// TwinCAT 3 PLC project CFFwelding
// ProgramVersion: 3.1.4024.0
// libraries:
//   Tc2_Standard, * (Beckhoff Automation GmbH)
//   Tc2_System, * (Beckhoff Automation GmbH)
//   Tc3_Module, * (Beckhoff Automation GmbH)
//   Tc2_MC2,3.3.65.0,Beckhoff Automation GmbH
// project tree:
//   Tasks/ Task_CffFast.TcTTO, Task_CffMain.TcTTO, Task_CffSlow.TcTTO
//   DUTs/Enums/ E_OperationMode.TcDUT, E_ControlSource.TcDUT, E_MachineState.TcDUT (not stored), E_InitializeState.TcDUT, E_MaintenanceFunction.TcDUT (not stored), E_MaintenanceState.TcDUT, E_CffState.TcDUT (not stored), E_CffExitIntent.TcDUT, E_CffStep.TcDUT, E_StepSubPhase.TcDUT, E_StepPrimaryCriterion.TcDUT, E_SecondaryCriterionAction.TcDUT, E_StepEndCause.TcDUT, E_ZCommandOwner.TcDUT, E_ZExtSetpointState.TcDUT (not stored), E_ZExternalTrajectoryState.TcDUT (not stored), E_AlarmLevel.TcDUT, E_AlarmCode.TcDUT (not stored), E_FastenerStatus.TcDUT, E_FeederState.TcDUT, E_ReturnMode.TcDUT, E_CalibrationState.TcDUT, E_CommandExecutionState.TcDUT, E_CommandRejectReason.TcDUT (not stored), E_HmiCommandCode.TcDUT, E_RobotCommandCode.TcDUT, E_ProgramState.TcDUT, E_InterfaceEventState.TcDUT
//   DUTs/Structures/ ST_MachineConfig.TcDUT (not stored), ST_MachineLimits.TcDUT (not stored), ST_ForceCalibration.TcDUT (not stored), ST_DisplacementCalibration.TcDUT, ST_CollisionCalibration.TcDUT (not stored), ST_ZForceControlProfile.TcDUT, ST_RAxisProfile.TcDUT (not stored), ST_StepProceedingConfig.TcDUT, ST_CffStepProgram.TcDUT (not stored), ST_JoinProgramHeader.TcDUT (not stored), ST_ProcessMonitorProfile.TcDUT, ST_CffJoinProgram.TcDUT (not stored), ST_JoiningPointAssignment.TcDUT, ST_CycleSnapshot.TcDUT, ST_ProcessActual.TcDUT (not stored), ST_ProcessFeatures.TcDUT, ST_StepCriterionResult.TcDUT, ST_CycleResult.TcDUT, ST_AlarmRequest.TcDUT (not stored), ST_AlarmStatus.TcDUT, ST_CommandMailbox.TcDUT, ST_CommandPermission.TcDUT, ST_MaintenanceHoldRequest.TcDUT, ST_RobotCommand.TcDUT (not stored), ST_RobotStatus.TcDUT, ST_FeederInput.TcDUT (not stored), ST_FeederOutput.TcDUT, ST_CalibrationCommand.TcDUT (not stored), ST_CalibrationStatus.TcDUT, ST_FastCommand.TcDUT (not stored), ST_FastStatus.TcDUT, ST_CurveSample.TcDUT, ST_HardwareBindingStatus.TcDUT (not stored), ST_SensorProcessingConfig.TcDUT (not stored), ST_ZExtSetpointConfig.TcDUT, ST_CffSequenceConfig.TcDUT, ST_CffFastConfigSnapshot.TcDUT (not stored)
//   GVLs/ GVL_Const.TcGVL (not stored), GVL_IO.TcGVL, GVL_Config.TcGVL, GVL_Calibration.TcGVL, GVL_Program.TcGVL, GVL_Command.TcGVL, GVL_Status.TcGVL, GVL_Process.TcGVL, GVL_Alarm.TcGVL, GVL_HMI.TcGVL (not stored), GVL_Trace.TcGVL, GVL_Persistent.TcGVL, GVL_ProjectInfo.TcGVL (not stored), GVL_FastInternal.TcGVL
//   DUTs/Interfaces/ ST_ZForceControlInput.TcDUT (not stored), ST_ZForceControlOutput.TcDUT, ST_ZExtSetpointCommand.TcDUT (not stored), ST_ZExtSetpointStatus.TcDUT, ST_ZAxisCommand.TcDUT, ST_ZAxisStatus.TcDUT, ST_RAxisCommand.TcDUT, ST_RAxisStatus.TcDUT (not stored), ST_CffMotionIntent.TcDUT (not stored), ST_ZExternalTrajectoryInput.TcDUT (not stored), ST_ZExternalTrajectoryOutput.TcDUT, ST_ContactDetectInput.TcDUT, ST_ContactDetectOutput.TcDUT, ST_ForceDeclineInput.TcDUT, ST_ForceDeclineOutput.TcDUT, ST_StepCriterionInput.TcDUT (not stored), ST_StepCriterionOutput.TcDUT, ST_CffSequenceCommand.TcDUT, ST_CffSequenceStatus.TcDUT (not stored), ST_ProcessReferenceCommand.TcDUT (not stored)
//   POUs/Functions/ FC_ClampLReal.TcPOU, FC_ScaleLinear.TcPOU (not stored), FC_LimitRate.TcPOU, FC_TrapezoidIntegrate.TcPOU (not stored), FC_RpmToRadPerSec.TcPOU (not stored), FC_CalcEnergyIncrement.TcPOU, FC_ConvertDirection.TcPOU, FC_IsFiniteLReal.TcPOU, FC_IsNewerRequestId.TcPOU (not stored), FC_ValidateCffSequenceConfig.TcPOU (not stored), FC_Interpolate1D.TcPOU, FC_ValidateCalibration.TcPOU, FC_ValidateJoinProgram.TcPOU, FC_GetPrimaryEndCause.TcPOU (not stored), FC_CalcStrokeVelocityLimit.TcPOU, FC_CheckModeSourceMatrix.TcPOU
//   POUs/FunctionBlocks/Utility/ FB_LowPassFilter.TcPOU, FB_Debounce.TcPOU (not stored), FB_SignalValidity.TcPOU (not stored), FB_SetpointRamp.TcPOU, FB_CommandHandshake.TcPOU, FB_AlarmLatch.TcPOU
//   POUs/FunctionBlocks/Axis/ FB_AxisCommandArbiter.TcPOU, FB_ZAxisNcAdapter.TcPOU, FB_RAxisNcAdapter.TcPOU, FB_ZAxisExtSetpointAdapter.TcPOU
//   POUs/FunctionBlocks/Control/ FB_BumplessProfileSwitch.TcPOU, FB_ZForceAdmittance.TcPOU, FB_ZExternalTrajectory.TcPOU, FB_ContactDetect.TcPOU (not stored), FB_ForceDeclineObserver.TcPOU, FB_StepProceedingCriterion.TcPOU
//   POUs/Fast/ PRG_FastInputs.TcPOU, PRG_CffSequence.TcPOU, PRG_FastAxisControl.TcPOU, PRG_FastMonitoring.TcPOU
//   POUs/Main/ PRG_ModeControl.TcPOU, PRG_RobotInterface.TcPOU (not stored), PRG_CommandDispatcher.TcPOU, PRG_ProgramManager.TcPOU, PRG_InitializeControl.TcPOU, PRG_ServiceCalibration.TcPOU (not stored), PRG_MaintenanceControl.TcPOU, PRG_ManualControl.TcPOU (not stored), PRG_AutoControl.TcPOU, PRG_FastenerControl.TcPOU, PRG_FeederControl.TcPOU, PRG_ClampControl.TcPOU (not stored), PRG_MachineMain.TcPOU (not stored), PRG_AlarmControl.TcPOU, PRG_TowerLightControl.TcPOU (not stored)
//   POUs/Slow/ PRG_HmiAdsInterface.TcPOU (not stored), PRG_ResultTraceability.TcPOU (not stored), PRG_Statistics.TcPOU, PRG_Persistence.TcPOU (not stored)
// real-time tasks:
//   TASK Task_CffMain: cycle T#10ms, priority 20, ADS port 350
//   TASK Task_CffFast: cycle T#2ms, priority 10, ADS port 351
//   TASK Task_CffSlow: cycle T#50000us, priority 30, ADS port 352
// motion (NC):
//   TASK NC_Cff SAF: cycle T#2ms, priority 4, ADS port 501
//   TASK NC_Cff SVB: cycle T#10ms, priority 8, ADS port 511
//   AXIS Z_Axis_NC (id 1)
//     OtherSettings: AllowMotionCmdToSlave=true
//     encoder EncType=1
//     drive DrvType=5
//       Analog: TorqueSetpointScale=10, ScaleFactorActTorque=0.1
//       TimeComp: TaskDelayCycles=1
//     controller CtrType=1
//       CtrPara: PriorControlFactor=1
//         Observer: BandWidth=20
//   AXIS R_Axis_NC (id 2)
//     OtherSettings: AllowMotionCmdToSlave=true
//     encoder EncType=1
//     drive DrvType=5
//       Analog: TorqueSetpointScale=10, ScaleFactorActTorque=0.1
//       TimeComp: TaskDelayCycles=1
//     controller CtrType=1
//       CtrPara: PriorControlFactor=1
//         Observer: BandWidth=20
// variable links:
//   CFFwelding/CFFwelding Instance <-> NC_Cff SAF/Axes/R_Axis_NC
//     Task_CffFast Inputs/GVL_IO.R_axis.NcToPlc <-> Outputs/ToPlc
//     Task_CffFast Outputs/GVL_IO.R_axis.PlcToNc <-> Inputs/FromPlc
//   CFFwelding/CFFwelding Instance <-> NC_Cff SAF/Axes/Z_Axis_NC
//     Task_CffFast Inputs/GVL_IO.Z_axis.NcToPlc <-> Outputs/ToPlc
//     Task_CffFast Outputs/GVL_IO.Z_axis.PlcToNc <-> Inputs/FromPlc

CONFIGURATION CFFwelding
    RESOURCE PLC ON TwinCAT3
        TASK Task_CffFast(INTERVAL := T#2ms, PRIORITY := 10);
        TASK Task_CffMain(INTERVAL := T#10ms, PRIORITY := 20);
        TASK Task_CffSlow(INTERVAL := T#50000us, PRIORITY := 30);
        PROGRAM PRG_FastInputs WITH Task_CffFast : PRG_FastInputs;
        PROGRAM PRG_CffSequence WITH Task_CffFast : PRG_CffSequence;
        PROGRAM PRG_FastAxisControl WITH Task_CffFast : PRG_FastAxisControl;
        PROGRAM PRG_FastMonitoring WITH Task_CffFast : PRG_FastMonitoring;
        PROGRAM PRG_ModeControl WITH Task_CffMain : PRG_ModeControl;
        PROGRAM PRG_RobotInterface WITH Task_CffMain : PRG_RobotInterface;
        PROGRAM PRG_CommandDispatcher WITH Task_CffMain : PRG_CommandDispatcher;
        PROGRAM PRG_ProgramManager WITH Task_CffMain : PRG_ProgramManager;
        PROGRAM PRG_InitializeControl WITH Task_CffMain : PRG_InitializeControl;
        PROGRAM PRG_ServiceCalibration WITH Task_CffMain : PRG_ServiceCalibration;
        PROGRAM PRG_MaintenanceControl WITH Task_CffMain : PRG_MaintenanceControl;
        PROGRAM PRG_ManualControl WITH Task_CffMain : PRG_ManualControl;
        PROGRAM PRG_AutoControl WITH Task_CffMain : PRG_AutoControl;
        PROGRAM PRG_FastenerControl WITH Task_CffMain : PRG_FastenerControl;
        PROGRAM PRG_FeederControl WITH Task_CffMain : PRG_FeederControl;
        PROGRAM PRG_ClampControl WITH Task_CffMain : PRG_ClampControl;
        PROGRAM PRG_MachineMain WITH Task_CffMain : PRG_MachineMain;
        PROGRAM PRG_AlarmControl WITH Task_CffMain : PRG_AlarmControl;
        PROGRAM PRG_TowerLightControl WITH Task_CffMain : PRG_TowerLightControl;
        PROGRAM PRG_HmiAdsInterface WITH Task_CffSlow : PRG_HmiAdsInterface;
        PROGRAM PRG_ResultTraceability WITH Task_CffSlow : PRG_ResultTraceability;
        PROGRAM PRG_Statistics WITH Task_CffSlow : PRG_Statistics;
        PROGRAM PRG_Persistence WITH Task_CffSlow : PRG_Persistence;
    END_RESOURCE
END_CONFIGURATION

// ---- DUTs/Enums/E_OperationMode.TcDUT
TYPE E_OperationMode : (
    OP_MODE_INVALID := 0,
    OP_MODE_MAINTENANCE := 10,
    OP_MODE_MANUAL := 20,
    OP_MODE_AUTOMATIC := 30
); END_TYPE

// ---- DUTs/Enums/E_ControlSource.TcDUT
TYPE E_ControlSource : (
    CONTROL_SOURCE_INVALID := 0,
    CONTROL_SOURCE_LOCAL := 10,
    CONTROL_SOURCE_ROBOT := 20
); END_TYPE

// ---- DUTs/Enums/E_InitializeState.TcDUT
TYPE E_InitializeState : (
    INIT_IDLE := 0,
    INIT_CLEAR_TRANSIENTS := 10,
    INIT_VALIDATE_MODE_SOURCE := 20,
    INIT_VALIDATE_COMMUNICATION := 30,
    INIT_VALIDATE_SENSORS := 40,
    INIT_RESET_AXIS_ERRORS := 50,
    INIT_HOME_Z_IF_REQUIRED := 60,
    INIT_HOME_R_IF_REQUIRED := 70,
    INIT_STOP_R := 80,
    INIT_RETURN_Z_REFERENCE := 90,
    INIT_RETURN_CYLINDERS := 100,
    INIT_RESET_FEEDER := 110,
    INIT_VALIDATE_CALIBRATIONS := 120,
    INIT_VALIDATE_ACTIVE_PROGRAM := 130,
    INIT_FINAL_READY_CHECK := 140,
    INIT_COMPLETE := 150,
    INIT_FAILED := 200
); END_TYPE

// ---- DUTs/Enums/E_MaintenanceState.TcDUT
TYPE E_MaintenanceState : (
    MAINT_STATE_IDLE := 0,
    MAINT_STATE_SELECTED := 10,
    MAINT_STATE_PRECHECK := 20,
    MAINT_STATE_ACTIVE := 30,
    MAINT_STATE_STOPPING := 40,
    MAINT_STATE_COMPLETE := 50,
    MAINT_STATE_CANCELLED := 60,
    MAINT_STATE_FAULT := 100
); END_TYPE

// ---- DUTs/Enums/E_CffExitIntent.TcDUT
TYPE E_CffExitIntent : (
    CFF_EXIT_NONE := 0,
    CFF_EXIT_NORMAL_RETURN := 10,
    CFF_EXIT_NOK_RETURN := 20,
    CFF_EXIT_ABORT_NO_RETURN := 30,
    CFF_EXIT_FAULT_NO_RETURN := 40
); END_TYPE

// ---- DUTs/Enums/E_CffStep.TcDUT
TYPE E_CffStep : (
    CFF_STEP_NONE := 0,
    CFF_STEP1_PENETRATION := 10,
    CFF_STEP2_CLEAN_ACTIVATE := 20,
    CFF_STEP3_WELDING := 30,
    CFF_STEP4_COMPRESSION := 40
); END_TYPE

// ---- DUTs/Enums/E_StepSubPhase.TcDUT
TYPE E_StepSubPhase : (
    STEP_SUBPHASE_NONE := 0,
    STEP_SUBPHASE_ENTRY := 10,
    STEP_SUBPHASE_RAMP_PROCESS := 20,
    STEP_SUBPHASE_END_CHECK := 30,
    STEP_SUBPHASE_BRAKE_COMPRESSION := 40,
    STEP_SUBPHASE_VALID_FORCE_HOLD := 50
); END_TYPE

// ---- DUTs/Enums/E_StepPrimaryCriterion.TcDUT
TYPE E_StepPrimaryCriterion : (
    STEP_CRIT_RELATIVE_DISTANCE := 0,
    STEP_CRIT_STEP_TIME := 10,
    STEP_CRIT_FORCE_DECLINE_TO := 20
); END_TYPE

// ---- DUTs/Enums/E_SecondaryCriterionAction.TcDUT
TYPE E_SecondaryCriterionAction : (
    SECONDARY_ADVANCE_AND_NOK := 0,
    SECONDARY_CONTROLLED_EXIT_NOK := 10
); END_TYPE

// ---- DUTs/Enums/E_StepEndCause.TcDUT
TYPE E_StepEndCause : (
    STEP_END_NONE := 0,
    STEP_END_PRIMARY_RELATIVE_DISTANCE := 10,
    STEP_END_PRIMARY_STEP_TIME := 20,
    STEP_END_PRIMARY_FORCE_DECLINE := 30,
    STEP_END_SECONDARY_RELATIVE_DISTANCE := 40,
    STEP_END_MAX_TIME := 50,
    STEP_END_HARD_FORCE := 60,
    STEP_END_HARD_STROKE := 70,
    STEP_END_COLLISION := 110,
    STEP_END_SENSOR_INVALID := 80,
    STEP_END_AXIS_FAULT := 90,
    STEP_END_STOP_REQUEST := 100
); END_TYPE

// ---- DUTs/Enums/E_ZCommandOwner.TcDUT
TYPE E_ZCommandOwner : (
    Z_OWNER_NONE := 0,
    Z_OWNER_HOME := 10,
    Z_OWNER_MANUAL := 20,
    Z_OWNER_APPROACH := 30,
    Z_OWNER_FORCE_PROCESS := 40,
    Z_OWNER_RETRACT := 50,
    Z_OWNER_FAULT_STOP := 100
); END_TYPE

// ---- DUTs/Enums/E_AlarmLevel.TcDUT
TYPE E_AlarmLevel : (
    ALARM_LEVEL_NONE := 0,
    ALARM_LEVEL_WARNING := 10,
    ALARM_LEVEL_NOK := 20,
    ALARM_LEVEL_FAULT := 30
); END_TYPE

// ---- DUTs/Enums/E_FastenerStatus.TcDUT
TYPE E_FastenerStatus : (
    FASTENER_UNKNOWN := 0,
    FASTENER_EMPTY := 10,
    FASTENER_SINGLE_OK := 20,
    FASTENER_WRONG_TYPE := 30,
    FASTENER_MULTIPLE := 40,
    FASTENER_JAMMED := 50,
    FASTENER_FAULT := 100
); END_TYPE

// ---- DUTs/Enums/E_FeederState.TcDUT
TYPE E_FeederState : (
    FEEDER_IDLE := 0,
    FEEDER_REQUEST := 10,
    FEEDER_FEEDING := 20,
    FEEDER_VERIFY := 30,
    FEEDER_COMPLETE := 40,
    FEEDER_FAULT := 100
); END_TYPE

// ---- DUTs/Enums/E_ReturnMode.TcDUT
TYPE E_ReturnMode : (
    RETURN_MODE_LOCAL := 0,
    RETURN_MODE_REFERENCE := 10
); END_TYPE

// ---- DUTs/Enums/E_CalibrationState.TcDUT
TYPE E_CalibrationState : (
    CAL_STATE_IDLE := 0,
    CAL_STATE_PRECHECK := 10,
    CAL_STATE_ACTIVE := 20,
    CAL_STATE_VALIDATE := 30,
    CAL_STATE_COMPLETE := 40,
    CAL_STATE_FAILED := 100
); END_TYPE

// ---- DUTs/Enums/E_CommandExecutionState.TcDUT
TYPE E_CommandExecutionState : (
    COMMAND_IDLE := 0,
    COMMAND_ACCEPTED := 10,
    COMMAND_EXECUTING := 20,
    COMMAND_COMPLETED := 30,
    COMMAND_REJECTED := 40,
    COMMAND_FAILED := 50,
    COMMAND_CANCELLED := 60
); END_TYPE

// ---- DUTs/Enums/E_HmiCommandCode.TcDUT
TYPE E_HmiCommandCode : (
    HMI_CMD_NONE := 0,
    HMI_CMD_START := 10,
    HMI_CMD_STOP := 20,
    HMI_CMD_INITIALIZE := 30,
    HMI_CMD_RESET := 40,
    HMI_CMD_ACK_RESULT := 50,
    HMI_CMD_SELECT_MAINTENANCE := 60,
    HMI_CMD_EXECUTE_MAINTENANCE := 70,
    HMI_CMD_CANCEL_MAINTENANCE := 80,
    HMI_CMD_VALIDATE_STEP := 90,
    HMI_CMD_SAVE_STEP := 100,
    HMI_CMD_VALIDATE_PROGRAM := 110,
    HMI_CMD_SAVE_PROGRAM := 120,
    HMI_CMD_ACTIVATE_PROGRAM := 130,
    HMI_CMD_SAVE_JOINING_POINT := 140,
    HMI_CMD_REQUEST_ALARM_PAGE := 150,
    HMI_CMD_REQUEST_CURVE_PAGE := 160
); END_TYPE

// ---- DUTs/Enums/E_RobotCommandCode.TcDUT
TYPE E_RobotCommandCode : (
    ROBOT_CMD_NONE := 0,
    ROBOT_CMD_START := 10,
    ROBOT_CMD_STOP := 20,
    ROBOT_CMD_INITIALIZE := 30,
    ROBOT_CMD_RESET := 40,
    ROBOT_CMD_ABORT := 50
); END_TYPE

// ---- DUTs/Enums/E_ProgramState.TcDUT
TYPE E_ProgramState : (
    PROGRAM_EMPTY := 0,
    PROGRAM_DRAFT := 10,
    PROGRAM_VALID := 20,
    PROGRAM_ACTIVE := 30,
    PROGRAM_INVALID := 40
); END_TYPE

// ---- DUTs/Enums/E_InterfaceEventState.TcDUT
TYPE E_InterfaceEventState : (
    INTERFACE_EVENT_IDLE := 0,
    INTERFACE_EVENT_CANDIDATE := 10,
    INTERFACE_EVENT_CONFIRMED := 20,
    INTERFACE_EVENT_REJECTED := 30,
    INTERFACE_EVENT_EXPIRED := 40
); END_TYPE

// ---- DUTs/Structures/ST_DisplacementCalibration.TcDUT
TYPE ST_DisplacementCalibration : STRUCT
    (* 位移传感器零点原始值。 *)
    fRawZero : LREAL;
    (* 原始值至毫米的增益。 *)
    fGainMmPerCount : LREAL;
    (* 位移零点偏置，单位毫米。 *)
    fOffsetMm : LREAL;
    (* 位移方向系数，仅允许正一或负一。 *)
    nDirection : DINT;
    (* 标定最大残差，单位毫米。 *)
    fMaxResidualMm : LREAL;
    (* 标定修订号。 *)
    nRevision : UDINT;
    (* 标定数据是否有效。 *)
    bValid : BOOL;
END_STRUCT
END_TYPE

// ---- DUTs/Structures/ST_ZForceControlProfile.TcDUT
TYPE ST_ZForceControlProfile : STRUCT
    (* Profile编号。 *)
    nProfileId : UDINT;
    (* Profile修订号；变化时必须执行积分无扰预置。 *)
    nRevision : UDINT;
    (* 速度前馈，向下为正，单位毫米每秒。 *)
    fVelocityFeedForwardMmS : LREAL;
    (* 比例增益，单位毫米每秒每千牛。 *)
    fKp : LREAL;
    (* 积分增益，单位毫米每二次方秒每千牛。 *)
    fKi : LREAL;
    (* 抗积分饱和回算增益，单位每秒。 *)
    fKaw : LREAL;
    (* 积分项绝对限幅，单位毫米每秒。 *)
    fIntegralLimit : LREAL;
    (* 向上最大速度，单位毫米每秒。 *)
    fMaxUpVelocityMmS : LREAL;
    (* 向下最大速度，单位毫米每秒。 *)
    fMaxDownVelocityMmS : LREAL;
    (* 最大加速度，单位毫米每二次方秒。 *)
    fMaxAccelerationMmS2 : LREAL;
    (* 制动距离裕量，单位毫米。 *)
    fBrakeMarginMm : LREAL;
    (* 设定力斜坡，单位牛顿每秒。 *)
    fForceRampNS : LREAL;
    (* 参数是否有效。 *)
    bValid : BOOL;
END_STRUCT
END_TYPE

// ---- DUTs/Structures/ST_StepProceedingConfig.TcDUT
TYPE ST_StepProceedingConfig : STRUCT
    (* 本步骤唯一主结束判据。 *)
    ePrimaryCriterion : E_StepPrimaryCriterion;
    (* 次级判据触发后的动作。 *)
    eSecondaryAction : E_SecondaryCriterionAction;
    (* 相对位移阈值，单位毫米。 *)
    fRelativeDistanceMm : LREAL;
    (* Step Time主判据目标，单位毫秒。 *)
    nPrimaryStepTimeMs : UDINT;
    (* 步骤质量最短时间，单位毫秒。 *)
    nStepMinMs : UDINT;
    (* Primary等待看门狗时间，单位毫秒。 *)
    nStepMaxMs : UDINT;
    (* Time或Decline主判据使用的累计S_rel次级边界，单位毫米。 *)
    fSecondarySRelMm : LREAL;
    (* 力下降确认阈值，单位牛顿。 *)
    fDeclineToN : LREAL;
    (* 力下降观察武装阈值，单位牛顿。 *)
    fArmForceN : LREAL;
    (* 力下降确认回差，单位牛顿。 *)
    fDeclineHysteresisN : LREAL;
    (* 力下降最小变化率绝对值，单位牛顿每秒。 *)
    fMinimumDeclineRateNS : LREAL;
    (* 力下降连续确认时间，单位毫秒。 *)
    nDeclineDebounceMs : UDINT;
    (* 力下降判据有效S_rel窗口下限，单位毫米。 *)
    fCriterionSRelMinMm : LREAL;
    (* 力下降判据有效S_rel窗口上限，单位毫米。 *)
    fCriterionSRelMaxMm : LREAL;
    (* 力下降判据最小主轴转速绝对值，单位转每分钟。 *)
    fCriterionRpmMin : LREAL;
    (* 判据允许的最大Z轴捕获速度绝对值，单位毫米每秒。 *)
    fCaptureMaxVelocityMmS : LREAL;
    (* 合格力带连续保持时间，单位毫秒。 *)
    nQualifiedForceHoldMs : UDINT;
    (* 合格力带容差，单位牛顿。 *)
    fForceBandToleranceN : LREAL;
    (* R轴停止阈值，单位转每分钟。 *)
    fRpmStoppedThresholdRpm : LREAL;
    (* 判据配置是否有效。 *)
    bValid : BOOL;
END_STRUCT
END_TYPE

// ---- DUTs/Structures/ST_ProcessMonitorProfile.TcDUT
TYPE ST_ProcessMonitorProfile : STRUCT
    (* 最小允许过程力，单位牛顿。 *)
    fMinForceN : LREAL;
    (* 最大允许过程力，单位牛顿。 *)
    fMaxForceN : LREAL;
    (* 最小允许相对位移，单位毫米。 *)
    fMinRelativeDistanceMm : LREAL;
    (* 最大允许相对位移，单位毫米。 *)
    fMaxRelativeDistanceMm : LREAL;
    (* 最小允许扭矩，单位牛米。 *)
    fMinTorqueNm : LREAL;
    (* 最大允许扭矩，单位牛米。 *)
    fMaxTorqueNm : LREAL;
    (* 最小允许能量，单位焦耳。 *)
    fMinEnergyJ : LREAL;
    (* 最大允许能量，单位焦耳。 *)
    fMaxEnergyJ : LREAL;
    (* 监控参数是否有效。 *)
    bValid : BOOL;
END_STRUCT
END_TYPE

// ---- DUTs/Structures/ST_JoiningPointAssignment.TcDUT
TYPE ST_JoiningPointAssignment : STRUCT
    (* 机器人加工点编号。 *)
    nJoiningPointId : UDINT;
    (* 该点关联的加工程序编号。 *)
    nProgramId : UDINT;
    (* 关联关系修订号。 *)
    nRevision : UDINT;
    (* 关联关系是否有效。 *)
    bValid : BOOL;
END_STRUCT
END_TYPE

// ---- DUTs/Structures/ST_CycleSnapshot.TcDUT
TYPE ST_CycleSnapshot : STRUCT
    (* 周期请求编号。 *)
    nRequestId : UDINT;
    (* 已接受的加工点编号。 *)
    nJoiningPointId : UDINT;
    (* 已冻结的加工程序。 *)
    stProgram : ST_CffJoinProgram;
    (* 机器配置修订号。 *)
    nMachineConfigRevision : UDINT;
    (* 标定修订号。 *)
    nCalibrationRevision : UDINT;
    (* 快照修订号。 *)
    nSnapshotRevision : UDINT;
    (* 快照完整性校验值。 *)
    nCrc32 : UDINT;
    (* 周期快照是否可执行。 *)
    bValid : BOOL;
END_STRUCT
END_TYPE

// ---- DUTs/Structures/ST_ProcessFeatures.TcDUT
TYPE ST_ProcessFeatures : STRUCT
    (* 周期最大力，单位牛顿。 *)
    fMaxForceN : LREAL;
    (* 周期平均力，单位牛顿。 *)
    fMeanForceN : LREAL;
    (* 周期最大扭矩，单位牛米。 *)
    fMaxTorqueNm : LREAL;
    (* 周期平均扭矩，单位牛米。 *)
    fMeanTorqueNm : LREAL;
    (* 周期最终相对位移，单位毫米。 *)
    fFinalRelativeDistanceMm : LREAL;
    (* 周期累计能量，单位焦耳。 *)
    fEnergyJ : LREAL;
    (* 有效采样数量。 *)
    nSampleCount : UDINT;
    (* 特征提取结果是否有效。 *)
    bValid : BOOL;
END_STRUCT
END_TYPE

// ---- DUTs/Structures/ST_StepCriterionResult.TcDUT
TYPE ST_StepCriterionResult : STRUCT
    (* 被评估的 CFF 步骤。 *)
    eStep : E_CffStep;
    (* 实际步骤结束原因。 *)
    eEndCause : E_StepEndCause;
    (* 主判据是否已经锁存。 *)
    bPrimaryLatched : BOOL;
    (* 次级判据是否已经锁存。 *)
    bSecondaryLatched : BOOL;
    (* 步骤是否判为不合格。 *)
    bNok : BOOL;
    (* 判据触发时的周期计数。 *)
    nTriggerCycle : UDINT;
    (* 步骤是否过短。 *)
    bTooShort : BOOL;
    (* 合格力带保持时间是否满足。 *)
    bQualifiedForceHoldMet : BOOL;
    (* 合格力带实际保持时间，单位秒。 *)
    rQualifiedForceHoldTime_s : LREAL;
    (* 锁存的轴向力，单位千牛。 *)
    rLatchedForce_kN : LREAL;
    (* 锁存的相对位置，单位毫米。 *)
    rLatchedRelativePosition_mm : LREAL;
    (* 锁存的步骤时间，单位秒。 *)
    rLatchedStepTime_s : LREAL;
END_STRUCT
END_TYPE

// ---- DUTs/Structures/ST_CycleResult.TcDUT
TYPE ST_CycleResult : STRUCT
    (* 全局焊接结果编号。 *)
    nWeldId : ULINT;
    (* 加工点编号。 *)
    nJoiningPointId : UDINT;
    (* 加工程序编号。 *)
    nProgramId : UDINT;
    (* 周期是否合格。 *)
    bOk : BOOL;
    (* 周期是否不合格。 *)
    bNok : BOOL;
    (* 周期是否中止。 *)
    bAborted : BOOL;
    (* 四个步骤的实际结束原因。 *)
    aeStepEndCause : ARRAY[1..4] OF E_StepEndCause;
    (* 周期特征值。 *)
    stFeatures : ST_ProcessFeatures;
    (* 周期持续时间，单位毫秒。 *)
    nCycleTimeMs : UDINT;
    (* 曲线缓冲区是否完整。 *)
    bCurveBufferComplete : BOOL;
    (* 已记录的曲线样本数量。 *)
    nCurveSampleCount : UDINT;
END_STRUCT
END_TYPE

// ---- DUTs/Structures/ST_AlarmStatus.TcDUT
TYPE ST_AlarmStatus : STRUCT
    (* 当前最高优先级报警代码。 *)
    eCurrentCode : E_AlarmCode;
    (* 当前最高报警等级。 *)
    eCurrentLevel : E_AlarmLevel;
    (* 是否存在活动报警。 *)
    bActive : BOOL;
    (* 当前报警是否已确认。 *)
    bAcknowledged : BOOL;
    (* 活动报警数量。 *)
    nActiveCount : UINT;
    (* 报警集合修订号。 *)
    nRevision : UDINT;
END_STRUCT
END_TYPE

// ---- DUTs/Structures/ST_CommandMailbox.TcDUT
TYPE ST_CommandMailbox : STRUCT
    (* 单调递增的命令请求编号。 *)
    nRequestId : UDINT;
    (* 控制源类型。 *)
    eSource : E_ControlSource;
    (* HMI 命令代码。 *)
    eHmiCommand : E_HmiCommandCode;
    (* 机器人命令代码。 *)
    eRobotCommand : E_RobotCommandCode;
    (* 命令目标对象编号。 *)
    nObjectId : UDINT;
    (* 通用整数载荷。 *)
    nPayloadDint : DINT;
    (* 通用浮点载荷。 *)
    fPayloadLreal : LREAL;
    (* 命令执行状态。 *)
    eState : E_CommandExecutionState;
    (* 命令拒绝原因。 *)
    eRejectReason : E_CommandRejectReason;
END_STRUCT
END_TYPE

// ---- DUTs/Structures/ST_CommandPermission.TcDUT
TYPE ST_CommandPermission : STRUCT
    (* 是否允许启动自动周期。 *)
    bAllowCycleStart : BOOL;
    (* 是否允许复位故障。 *)
    bAllowReset : BOOL;
    (* 是否允许手动 Z 轴动作。 *)
    bAllowManualZ : BOOL;
    (* 是否允许手动 R 轴动作。 *)
    bAllowManualR : BOOL;
    (* 是否允许执行维护功能。 *)
    bAllowMaintenance : BOOL;
    (* 是否允许执行标定。 *)
    bAllowCalibration : BOOL;
    (* 禁止原因位掩码。 *)
    nInhibitMask : UDINT;
END_STRUCT
END_TYPE

// ---- DUTs/Structures/ST_MaintenanceHoldRequest.TcDUT
TYPE ST_MaintenanceHoldRequest : STRUCT
    (* 维护请求编号。 *)
    nRequestId : UDINT;
    (* 请求的维护功能。 *)
    eFunction : E_MaintenanceFunction;
    (* 请求保持的目标力，单位牛顿。 *)
    fHoldForceN : LREAL;
    (* 最大保持时间，单位毫秒。 *)
    nTimeoutMs : UDINT;
    (* 请求是否有效。 *)
    bExecute : BOOL;
    (* 请求是否取消。 *)
    bCancel : BOOL;
END_STRUCT
END_TYPE

// ---- DUTs/Structures/ST_RobotStatus.TcDUT
TYPE ST_RobotStatus : STRUCT
    (* 已接受的机器人命令序号。 *)
    nAcceptedSequence : UDINT;
    (* 机器是否准备好接收命令。 *)
    bReady : BOOL;
    (* 机器是否正在执行命令。 *)
    bBusy : BOOL;
    (* 最近命令是否完成。 *)
    bComplete : BOOL;
    (* 最近周期是否合格。 *)
    bOk : BOOL;
    (* 最近周期是否不合格。 *)
    bNok : BOOL;
    (* 机器是否存在故障。 *)
    bFault : BOOL;
    (* 已接受的加工点编号。 *)
    nAcceptedJoiningPointId : UDINT;
    (* 最近焊接结果编号。 *)
    nWeldId : ULINT;
    (* 最近命令拒绝原因。 *)
    eRejectReason : E_CommandRejectReason;
END_STRUCT
END_TYPE

// ---- DUTs/Structures/ST_FeederOutput.TcDUT
TYPE ST_FeederOutput : STRUCT
    (* 请求供给一个紧固件。 *)
    bFeedRequest : BOOL;
    (* 请求停止供料器。 *)
    bStop : BOOL;
    (* 请求复位供料器故障。 *)
    bReset : BOOL;
    (* 供料模式编号。 *)
    nMode : UINT;
END_STRUCT
END_TYPE

// ---- DUTs/Structures/ST_CalibrationStatus.TcDUT
TYPE ST_CalibrationStatus : STRUCT
    (* 已接受的标定请求编号。 *)
    nAcceptedRequestId : UDINT;
    (* 标定状态。 *)
    eState : E_CalibrationState;
    (* 标定是否完成。 *)
    bDone : BOOL;
    (* 标定是否发生错误。 *)
    bError : BOOL;
    (* 标定错误原因编号。 *)
    nErrorReason : UDINT;
    (* 生成的标定修订号。 *)
    nRevision : UDINT;
END_STRUCT
END_TYPE

// ---- DUTs/Structures/ST_FastStatus.TcDUT
TYPE ST_FastStatus : STRUCT
    (* 快速任务已接受的命令请求编号。 *)
    nAcceptedRequestId : UDINT;
    (* 快速任务循环计数。 *)
    nCycleCounter : UDINT;
    (* 快速任务实际周期，单位微秒。 *)
    nActualPeriodUs : UDINT;
    (* CFF 顺序状态。 *)
    stSequence : ST_CffSequenceStatus;
    (* Z 轴状态。 *)
    stZAxis : ST_ZAxisStatus;
    (* Z轴External Setpoint生命周期状态。 *)
    stZExtSetpoint : ST_ZExtSetpointStatus;
    (* Z轴External轨迹状态。 *)
    stZExternalTrajectory : ST_ZExternalTrajectoryOutput;
    (* 已接受的Sequence Z轴命令事务号。 *)
    udiAcceptedSequenceZCommandId : UDINT;
    (* 已接受的Sequence R轴命令事务号。 *)
    udiAcceptedSequenceRCommandId : UDINT;
    (* Z轴导纳力控速度和Anti-windup诊断。 *)
    stZForceControl : ST_ZForceControlOutput;
    (* R 轴状态。 *)
    stRAxis : ST_RAxisStatus;
    (* R轴转速包络，单位转每分钟。 *)
    rRSpeedEnvelope_rpm : LREAL;
    (* R轴转速斜坡正在执行。 *)
    bRSpeedRampBusy : BOOL;
    (* R轴转速斜坡已经达到目标。 *)
    bRSpeedRampReached : BOOL;
    (* R轴转速斜坡参数有效。 *)
    bRSpeedRampValid : BOOL;
    (* 力设定值斜坡已经达到目标。 *)
    bForceSetpointRampReached : BOOL;
    (* 力设定值斜坡参数有效。 *)
    bForceSetpointRampValid : BOOL;
    (* 快速过程实际值。 *)
    stProcess : ST_ProcessActual;
END_STRUCT
END_TYPE

// ---- DUTs/Structures/ST_CurveSample.TcDUT
TYPE ST_CurveSample : STRUCT
    (* 快速任务循环计数。 *)
    nCycleCounter : UDINT;
    (* 单调时间戳，单位微秒。 *)
    nTimestampUs : ULINT;
    (* 过程力，单位牛顿。 *)
    fForceN : LREAL;
    (* 接触点后的相对位移，单位毫米。 *)
    fRelativeDistanceMm : LREAL;
    (* R 轴转速，单位转每分钟。 *)
    fSpeedRpm : LREAL;
    (* R 轴扭矩，单位牛米。 *)
    fTorqueNm : LREAL;
    (* 瞬时机械功率，单位瓦。 *)
    fPowerW : LREAL;
END_STRUCT
END_TYPE

// ---- DUTs/Structures/ST_ZExtSetpointConfig.TcDUT
TYPE ST_ZExtSetpointConfig : STRUCT
    (* External Setpoint配置已经过受控确认；默认FALSE禁止使能。 *)
    bValid : BOOL;
    (* 等待NC确认使能的最大时间。 *)
    tEnableTimeout : TIME;
    (* 等待NC确认禁用的最大时间。 *)
    tDisableTimeout : TIME;
    (* 判定速度已受控归零的绝对阈值，单位毫米每秒。 *)
    rStandstillVelocity_mm_s : LREAL;
    (* 相邻Feed允许的位置偏差上限，单位毫米。 *)
    rMaximumPositionDeviation_mm : LREAL;
    (* 相邻Feed允许的速度变化上限，单位毫米每秒。 *)
    rMaximumVelocityStep_mm_s : LREAL;
    (* 速度归零后保持最后非零Direction的Fast周期数，至少1。 *)
    nDirectionHoldCycles : UINT;
    (* Disable确认后继续保持零Feed的Fast周期数，至少1。 *)
    nPostDisableHoldCycles : UINT;
END_STRUCT
END_TYPE

// ---- DUTs/Structures/ST_CffSequenceConfig.TcDUT
TYPE ST_CffSequenceConfig : STRUCT
    (* Approach标准定位等待超时。 *)
    tApproachTimeout : TIME;
    (* External Contact Search等待超时。 *)
    tContactSearchTimeout : TIME;
    (* Contact参考点事务确认等待超时。 *)
    tContactReferenceAckTimeout : TIME;
    (* 受控卸载等待超时。 *)
    tControlledUnloadTimeout : TIME;
    (* 卸载静止条件连续确认时间。 *)
    tUnloadStandstillConfirm : TIME;
    (* R轴受控停止等待超时。 *)
    tRAxisStopTimeout : TIME;
    (* 标准NC返回等待超时。 *)
    tReturnTimeout : TIME;
    (* Approach和Return标准NC加速度，单位mm/s2。 *)
    fStandardMoveAccelerationMmS2 : LREAL;
    (* Approach和Return标准NC减速度，单位mm/s2。 *)
    fStandardMoveDecelerationMmS2 : LREAL;
    (* 配置已受控确认。 *)
    bValid : BOOL;
END_STRUCT
END_TYPE

// ---- DUTs/Interfaces/ST_ZForceControlOutput.TcDUT
TYPE ST_ZForceControlOutput :
STRUCT
    (* 导纳控制输出的Z轴速度命令，向下为正，单位mm/s。 *)
    rVelocityCommand_mm_s : LREAL;
    (* PI积分分量，单位mm/s，用于诊断Anti-windup。 *)
    rIntegralTerm_mm_s : LREAL;
    (* 斜坡后的目标力，单位kN。 *)
    rForceSetRamped_kN : LREAL;
    (* 目标力减ForceControl实际力，单位kN。 *)
    rForceError_kN : LREAL;
    (* 前馈、比例和积分相加后的未饱和速度，单位mm/s。 *)
    rUnsaturatedVelocity_mm_s : LREAL;
    (* 固定边界、加速度和最终S_rel包络限幅后的速度，单位mm/s。 *)
    rSaturatedVelocity_mm_s : LREAL;
    (* 当前S_rel剩余行程对应的向下制动速度上限，单位mm/s。 *)
    rStrokeVelocityLimit_mm_s : LREAL;
    (* 算法已使能并正在计算输出。 *)
    bActive : BOOL;
    (* 输出受到速度、位移、加速度或硬边界限制。 *)
    bLimited : BOOL;
    (* 当前周期按门控或硬边界冻结积分。 *)
    bAntiWindupFrozen : BOOL;
    (* Hard Force、Hard S_rel或Collision边界当前有效。 *)
    bHardLimitActive : BOOL;
    (* 算法输入无效或内部诊断失败。 *)
    bFault : BOOL;
    (* 算法故障编号，0表示无故障。 *)
    nFaultId : UDINT;
END_STRUCT
END_TYPE

// ---- DUTs/Interfaces/ST_ZExtSetpointStatus.TcDUT
TYPE ST_ZExtSetpointStatus :
STRUCT
    (* 外部设定值接口已经成功使能。 *)
    bEnabled : BOOL;
    (* 适配器正在执行使能、送值或禁用阶段。 *)
    bBusy : BOOL;
    (* 本次生命周期正常完成。 *)
    bDone : BOOL;
    (* 当前扫描成功写入P/V/A/Direction。 *)
    bFeedAccepted : BOOL;
    (* External已完整退出，允许Owner转交标准NC。 *)
    bReleaseOwner : BOOL;
    (* 运动控制接口或生命周期诊断报告错误。 *)
    bError : BOOL;
    (* 运动控制错误编号，零表示无错误。 *)
    nErrorId : UDINT;
    (* 外部设定值生命周期状态。 *)
    eState : E_ZExtSetpointState;
    (* 已执行的External Feed周期计数。 *)
    udiFeedCycleCounter : UDINT;
    (* 已接受设定值有效。 *)
    bAcceptedSetpointValid : BOOL;
    (* 已接受位置，单位mm。 *)
    rAcceptedPosition_mm : LREAL;
    (* 已接受速度，单位mm/s。 *)
    rAcceptedVelocity_mm_s : LREAL;
    (* 已接受加速度，单位mm/s2。 *)
    rAcceptedAcceleration_mm_s2 : LREAL;
    (* 已接受方向。 *)
    nAcceptedDirection : DINT;
END_STRUCT
END_TYPE

// ---- DUTs/Interfaces/ST_ZAxisCommand.TcDUT
TYPE ST_ZAxisCommand :
STRUCT
    (* 请求使能 Z 轴。 *)
    bEnable : BOOL;
    (* 请求复位 Z 轴错误。 *)
    bReset : BOOL;
    (* 请求受控停止 Z 轴。 *)
    bStop : BOOL;
    (* 请求执行标准 NC 回零。 *)
    bHome : BOOL;
    (* 请求标准绝对定位。 *)
    bMoveAbsolute : BOOL;
    (* 请求标准速度运动。 *)
    bMoveVelocity : BOOL;
    (* 请求由外部设定值适配器接管。 *)
    bUseExternalSetpoint : BOOL;
    (* 回零完成后使用的参考位置，向下为正，单位毫米。 *)
    rHomePosition_mm : LREAL;
    (* 绝对位置目标，向下为正，单位毫米。 *)
    rPosition_mm : LREAL;
    (* 速度目标，向下为正，单位毫米每秒。 *)
    rVelocity_mm_s : LREAL;
    (* 加速度限制，单位毫米每二次方秒。 *)
    rAcceleration_mm_s2 : LREAL;
    (* 减速度限制，单位毫米每二次方秒。 *)
    rDeceleration_mm_s2 : LREAL;
    (* 请求取得控制权的命令所有者。 *)
    eOwnerRequest : E_ZCommandOwner;
END_STRUCT
END_TYPE

// ---- DUTs/Interfaces/ST_ZAxisStatus.TcDUT
TYPE ST_ZAxisStatus :
STRUCT
    (* Z 轴程序接口具备接收命令的内部条件。 *)
    bReady : BOOL;
    (* Z 轴已经使能。 *)
    bEnabled : BOOL;
    (* Z 轴已完成回零并具有有效参考坐标。 *)
    bHomed : BOOL;
    (* Z 轴正在运动。 *)
    bMoving : BOOL;
    (* Z 轴处于静止状态。 *)
    bStandstill : BOOL;
    (* 标准 NC 命令仍在执行。 *)
    bBusy : BOOL;
    (* 最近标准 NC 命令已经完成。 *)
    bDone : BOOL;
    (* 外部设定值生命周期有效。 *)
    bExternalSetpointActive : BOOL;
    (* Z 轴适配器报告错误。 *)
    bError : BOOL;
    (* Z 轴或运动控制错误编号，零表示无错误。 *)
    nErrorId : UDINT;
    (* 当前唯一命令所有者。 *)
    eActiveOwner : E_ZCommandOwner;
    (* Z 轴 Adapter 已处理的最后命令事务编号。 *)
    udiAcceptedCommandId : UDINT;
    (* Z 轴实际位置，向下为正，单位毫米。 *)
    rActualPosition_mm : LREAL;
    (* Z 轴实际速度，向下为正，单位毫米每秒。 *)
    rActualVelocity_mm_s : LREAL;
END_STRUCT
END_TYPE

// ---- DUTs/Interfaces/ST_RAxisCommand.TcDUT
TYPE ST_RAxisCommand :
STRUCT
    (* 请求使能R轴。 *)
    bEnable : BOOL;
    (* 请求复位R轴错误。 *)
    bReset : BOOL;
    (* 请求受控停止R轴。 *)
    bStop : BOOL;
    (* 请求速度运行。 *)
    bMoveVelocity : BOOL;
    (* 摩擦主轴速度目标，单位rpm。 *)
    rVelocity_rpm : LREAL;
    (* 速度斜坡加速度，单位rpm/s。 *)
    rAcceleration_rpm_s : LREAL;
    (* 速度斜坡减速度，单位rpm/s。 *)
    rDeceleration_rpm_s : LREAL;
END_STRUCT
END_TYPE

// ---- DUTs/Interfaces/ST_ZExternalTrajectoryOutput.TcDUT
TYPE ST_ZExternalTrajectoryOutput : STRUCT
    (* 轨迹位置，单位mm。 *)
    rPosition_mm : LREAL;
    (* 轨迹速度，单位mm/s。 *)
    rVelocity_mm_s : LREAL;
    (* 轨迹加速度，单位mm/s2。 *)
    rAcceleration_mm_s2 : LREAL;
    (* 轨迹方向。 *)
    nDirection : DINT;
    (* 轨迹发生器状态。 *)
    eState : E_ZExternalTrajectoryState;
    (* 正在执行方向过渡。 *)
    bDirectionTransition : BOOL;
    (* 零速度已经确认。 *)
    bZeroConfirmed : BOOL;
    (* 正方向运动已禁止。 *)
    bPositiveMotionInhibited : BOOL;
    (* 轨迹发生器活动。 *)
    bActive : BOOL;
    (* 轨迹发生器故障。 *)
    bFault : BOOL;
    (* 轨迹发生器故障编号。 *)
    nFaultId : UDINT;
END_STRUCT
END_TYPE

// ---- DUTs/Interfaces/ST_ContactDetectInput.TcDUT
TYPE ST_ContactDetectInput :
STRUCT
    (* Contact检测使能请求。 *)
    bEnable : BOOL;
    (* Contact检测复位请求。 *)
    bReset : BOOL;
    (* 当前压向实际力，单位kN。 *)
    rForceActual_kN : LREAL;
    (* Contact候选置位力阈值，单位kN。 *)
    rForceOn_kN : LREAL;
    (* Contact候选释放力阈值，单位kN。 *)
    rForceOff_kN : LREAL;
    (* 当前Z轴位置，向下为正，单位mm。 *)
    rAxisPosition_mm : LREAL;
    (* 当前外部位移绝对值，单位mm。 *)
    rSensorPosition_mm : LREAL;
    (* Contact允许的Z轴绝对位置下限，单位mm。 *)
    rAxisPositionMinimum_mm : LREAL;
    (* Contact允许的Z轴绝对位置上限，单位mm。 *)
    rAxisPositionMaximum_mm : LREAL;
    (* Contact允许的外部位移绝对位置下限，单位mm。 *)
    rSensorPositionMinimum_mm : LREAL;
    (* Contact允许的外部位移绝对位置上限，单位mm。 *)
    rSensorPositionMaximum_mm : LREAL;
    (* 当前Z轴速度，向下为正，单位mm/s。 *)
    rAxisVelocity_mm_s : LREAL;
    (* Contact捕获允许的最大速度绝对值，单位mm/s。 *)
    rCaptureMaximumVelocity_mm_s : LREAL;
    (* Contact连续确认时间，单位s。 *)
    rDebounceTime_s : LREAL;
    (* 实际调用周期，单位s。 *)
    rCycleTime_s : LREAL;
    (* 输入采样有效。 *)
    bSignalValid : BOOL;
END_STRUCT
END_TYPE

// ---- DUTs/Interfaces/ST_ContactDetectOutput.TcDUT
TYPE ST_ContactDetectOutput :
STRUCT
    (* Force On已经形成尚未确认的Contact候选。 *)
    bCandidate : BOOL;
    (* Contact已经防抖确认。 *)
    bDetected : BOOL;
    (* Contact候选时锁存的压向力，单位kN。 *)
    rCandidateForce_kN : LREAL;
    (* Contact候选时锁存的Z轴绝对位置，单位mm。 *)
    rCandidateAxisPosition_mm : LREAL;
    (* Contact候选时锁存的外部位移绝对位置，单位mm。 *)
    rCandidateSensorPosition_mm : LREAL;
    (* Contact确认时锁存的压向力，单位kN。 *)
    rDetectedForce_kN : LREAL;
    (* Contact确认时锁存的Z轴绝对位置，单位mm。 *)
    rDetectedAxisPosition_mm : LREAL;
    (* Contact确认时锁存的外部位移绝对位置，单位mm。 *)
    rDetectedSensorPosition_mm : LREAL;
    (* Contact确认时仅一个扫描周期的参考点锁存请求。 *)
    bReferenceLatchRequest : BOOL;
    (* 输入无效或检测窗口异常。 *)
    bFault : BOOL;
    (* Contact故障编号，0表示无故障。 *)
    nFaultId : UDINT;
END_STRUCT
END_TYPE

// ---- DUTs/Interfaces/ST_ForceDeclineInput.TcDUT
TYPE ST_ForceDeclineInput :
STRUCT
    (* 力下降观察使能请求。 *)
    bEnable : BOOL;
    (* 清除观察器内部状态和故障。 *)
    bReset : BOOL;
    (* Force、RPM、S_rel、速度和周期均有效。 *)
    bSignalValid : BOOL;
    (* 当前判据力，单位kN。 *)
    rForceActual_kN : LREAL;
    (* 当前主轴转速，单位rpm。 *)
    rSpeed_rpm : LREAL;
    (* Contact起累计S_rel，单位mm。 *)
    rRelativePosition_mm : LREAL;
    (* 当前Z轴速度，向下为正，单位mm/s。 *)
    rAxisVelocity_mm_s : LREAL;
    (* 当前步骤累计时间，单位s。 *)
    rStepTime_s : LREAL;
    (* 力下降观察武装阈值，单位kN。 *)
    rArmForce_kN : LREAL;
    (* 力下降确认阈值，单位kN。 *)
    rDeclineTo_kN : LREAL;
    (* 力下降确认回差，单位kN。 *)
    rHysteresis_kN : LREAL;
    (* 最小下降率绝对值，单位kN/s。 *)
    rMinimumDeclineRate_kN_s : LREAL;
    (* 有效S_rel窗口下限，单位mm。 *)
    rCriterionSRelMinimum_mm : LREAL;
    (* 有效S_rel窗口上限，单位mm。 *)
    rCriterionSRelMaximum_mm : LREAL;
    (* 有效主轴转速绝对值下限，单位rpm。 *)
    rCriterionRpmMinimum : LREAL;
    (* 允许确认的Z轴速度绝对值上限，单位mm/s。 *)
    rCaptureMaximumVelocity_mm_s : LREAL;
    (* 连续确认时间，单位s。 *)
    rDebounceTime_s : LREAL;
    (* 实际调用周期，单位s。 *)
    rCycleTime_s : LREAL;
END_STRUCT
END_TYPE

// ---- DUTs/Interfaces/ST_ForceDeclineOutput.TcDUT
TYPE ST_ForceDeclineOutput :
STRUCT
    (* 当前步骤已经达到Arm Force。 *)
    bArmed : BOOL;
    (* 当前处于Decline回差候选窗口。 *)
    bCandidate : BOOL;
    (* Force Decline已经连续确认。 *)
    bConfirmed : BOOL;
    (* 相邻有效样本计算的力变化率，单位kN/s。 *)
    rForceDerivative_kN_s : LREAL;
    (* 当前连续确认累计时间，单位s。 *)
    rStableTime_s : LREAL;
    (* 确认时锁存的力，单位kN。 *)
    rLatchedForce_kN : LREAL;
    (* 确认时锁存的累计S_rel，单位mm。 *)
    rLatchedRelativePosition_mm : LREAL;
    (* 确认时锁存的主轴转速，单位rpm。 *)
    rLatchedSpeed_rpm : LREAL;
    (* 确认时锁存的步骤时间，单位s。 *)
    rLatchedStepTime_s : LREAL;
    (* 输入、配置或数值计算故障。 *)
    bFault : BOOL;
    (* 确定性故障编号，零表示无故障。 *)
    nFaultId : UDINT;
END_STRUCT
END_TYPE

// ---- DUTs/Interfaces/ST_StepCriterionOutput.TcDUT
TYPE ST_StepCriterionOutput :
STRUCT
    (* 力下降判据已经达到预装配力并进入可确认窗口。 *)
    bArmed : BOOL;
    (* 主判据已经满足。 *)
    bPrimaryMet : BOOL;
    (* 次级相对位移限制已经触发。 *)
    bSecondaryLimitReached : BOOL;
    (* 当前步骤结束已经防抖确认。 *)
    bEndConfirmed : BOOL;
    (* Primary满足时步骤时间低于StepMin。 *)
    bTooShort : BOOL;
    (* 当前结束原因要求周期或步骤判为不合格。 *)
    bNok : BOOL;
    (* Secondary AdvanceAndNok允许进入下一步骤。 *)
    bAdvanceRequested : BOOL;
    (* Secondary、StepMax或硬原因要求受控退出。 *)
    bControlledExitRequested : BOOL;
    (* 当前结束原因要求立即禁止继续向下。 *)
    bDownwardMotionInhibited : BOOL;
    (* 步骤实际结束原因。 *)
    eEndCause : E_StepEndCause;
    (* 结束确认时锁存的轴向力，单位千牛。 *)
    rLatchedForce_kN : LREAL;
    (* 结束确认时锁存的相对位移，单位毫米。 *)
    rLatchedRelativePosition_mm : LREAL;
    (* 结束确认时锁存的步骤时间，单位秒。 *)
    rLatchedStepTime_s : LREAL;
    (* 输入、配置或未知枚举故障。 *)
    bFault : BOOL;
    (* 确定性故障编号，零表示无故障。 *)
    nFaultId : UDINT;
END_STRUCT
END_TYPE

// ---- DUTs/Interfaces/ST_CffSequenceCommand.TcDUT
TYPE ST_CffSequenceCommand :
STRUCT
    (* 启动一次CFF循环的一次性内部脉冲。 *)
    bStartPulse : BOOL;
    (* 请求受控停止的一次性内部脉冲。 *)
    bStopPulse : BOOL;
    (* 请求立即退出流程的一次性内部脉冲。 *)
    bAbortPulse : BOOL;
    (* 请求复位流程锁存状态的一次性内部脉冲。 *)
    bResetPulse : BOOL;
    (* 已由命令仲裁接受的事务编号。 *)
    nCommandId : UDINT;
    (* 选择的焊接程序编号。 *)
    nProgramId : UDINT;
    (* 选择的Joining Point编号。 *)
    nJoiningPointId : UDINT;
    (* 生产硬件、模式和权限前置条件均有效。 *)
    bProductionPermission : BOOL;
END_STRUCT
END_TYPE

// ---- GVLs/GVL_IO.TcGVL
{attribute 'qualified_only'}
{attribute 'TcContextName' := 'Task_CffFast'}
VAR_GLOBAL
    (* Z 轴 PLC 运动控制引用；仅允许连接离线 NC 轴，不绑定真实驱动。 *)
    Z_axis : AXIS_REF;
    (* R 轴 PLC 运动控制引用；仅允许连接离线 NC 轴，不绑定真实驱动。 *)
    R_axis : AXIS_REF;

    (* TODO_HW_MAP：力传感器原始输入通道，当前未映射。 *)
    nForceChannelRaw AT %I* : INT;
    (* TODO_HW_MAP：EP3174力通道错误状态，当前未映射。 *)
    bForceChannelError AT %I* : BOOL;
    (* TODO_HW_MAP：EP3174力通道上溢状态，当前未映射。 *)
    bForceChannelOverrange AT %I* : BOOL;
    (* TODO_HW_MAP：EP3174力通道下溢状态，当前未映射。 *)
    bForceChannelUnderrange AT %I* : BOOL;
    (* TODO_HW_MAP：位移传感器原始输入通道，当前未映射。 *)
    nDisplacementChannelRaw AT %I* : INT;
    (* TODO_HW_MAP：位移输入通道错误状态，当前未映射。 *)
    bDisplacementChannelError AT %I* : BOOL;
    (* TODO_HW_MAP：位移输入通道上溢状态，当前未映射。 *)
    bDisplacementChannelOverrange AT %I* : BOOL;
    (* TODO_HW_MAP：位移输入通道下溢状态，当前未映射。 *)
    bDisplacementChannelUnderrange AT %I* : BOOL;
    (* TODO_HW_MAP：Collision Reference Sensor输入，当前未映射。 *)
    bCollisionReferenceSensor AT %I* : BOOL;
    (* TODO_HW_MAP：碰撞检测输入，当前未映射。 *)
    bCollisionDetected AT %I* : BOOL;
    (* TODO_HW_MAP：紧固件在位输入，当前未映射。 *)
    bFastenerPresent AT %I* : BOOL;
    (* TODO_HW_MAP：供料器就绪输入，当前未映射。 *)
    bFeederReady AT %I* : BOOL;
    (* TODO_HW_MAP：夹紧到位输入，当前未映射。 *)
    bClampClosed AT %I* : BOOL;
    (* TODO_HW_MAP：机器人许可输入，当前未映射。 *)
    bRobotPermit AT %I* : BOOL;

    (* TODO_HW_MAP：供料请求输出，当前未映射。 *)
    bFeedRequest AT %Q* : BOOL;
    (* TODO_HW_MAP：夹紧请求输出，当前未映射。 *)
    bClampRequest AT %Q* : BOOL;
    (* TODO_HW_MAP：机器人就绪输出，当前未映射。 *)
    bRobotReady AT %Q* : BOOL;
    (* TODO_HW_MAP：红色塔灯输出，当前未映射。 *)
    bTowerRed AT %Q* : BOOL;
    (* TODO_HW_MAP：黄色塔灯输出，当前未映射。 *)
    bTowerYellow AT %Q* : BOOL;
    (* TODO_HW_MAP：绿色塔灯输出，当前未映射。 *)
    bTowerGreen AT %Q* : BOOL;
END_VAR

// ---- GVLs/GVL_Config.TcGVL
{attribute 'qualified_only'}
VAR_GLOBAL
    (* 当前机器配置。 *)
    stMachine : ST_MachineConfig;
    (* 当前机器运动和过程限值。 *)
    stLimits : ST_MachineLimits;
    (* 当前 Z 轴力控制参数。 *)
    stZForceControl : ST_ZForceControlProfile;
    (* 当前 R 轴参数。 *)
    stRAxis : ST_RAxisProfile;
    (* 当前快速传感器滤波、范围和诊断参数。 *)
    stSensorProcessing : ST_SensorProcessingConfig;
    (* Z轴External Setpoint超时、连续性和退出保持参数。 *)
    stZExtSetpoint : ST_ZExtSetpointConfig;
    (* CFF流程超时和标准定位斜率；默认无效。 *)
    stCffSequence : ST_CffSequenceConfig;
END_VAR

// ---- GVLs/GVL_Calibration.TcGVL
{attribute 'qualified_only'}
VAR_GLOBAL
    (* 力传感器标定数据。 *)
    stForce : ST_ForceCalibration;
    (* 位移传感器标定数据。 *)
    stDisplacement : ST_DisplacementCalibration;
    (* 碰撞基准标定数据。 *)
    stCollision : ST_CollisionCalibration;
    (* 标定命令邮箱。 *)
    stCommand : ST_CalibrationCommand;
    (* 标定执行状态。 *)
    stStatus : ST_CalibrationStatus;
END_VAR

// ---- GVLs/GVL_Program.TcGVL
{attribute 'qualified_only'}
VAR_GLOBAL
    (* 加工程序数据库。 *)
    astJoinPrograms : ARRAY[1..64] OF ST_CffJoinProgram;
    (* 加工点至程序的关联数据库。 *)
    astJoiningPointAssignments : ARRAY[1..512] OF ST_JoiningPointAssignment;
    (* 当前周期冻结快照。 *)
    stCycleSnapshot : ST_CycleSnapshot;
    (* 已选择的程序编号。 *)
    nSelectedProgramId : UDINT;
END_VAR

// ---- GVLs/GVL_Command.TcGVL
{attribute 'qualified_only'}
VAR_GLOBAL
    (* 统一外部命令邮箱。 *)
    stMailbox : ST_CommandMailbox;
    (* 当前命令权限计算结果。 *)
    stPermission : ST_CommandPermission;
    (* CFF流程发布给快速输入层的Contact参考点事务。 *)
    stProcessReference : ST_ProcessReferenceCommand;
    (* 主任务发布给快速任务的命令。 *)
    stFast : ST_FastCommand;
    (* 机器人接口命令。 *)
    stRobot : ST_RobotCommand;
    (* 维护力保持请求。 *)
    stMaintenanceHold : ST_MaintenanceHoldRequest;
    (* 供料器输出命令。 *)
    stFeeder : ST_FeederOutput;
END_VAR

// ---- GVLs/GVL_Status.TcGVL
{attribute 'qualified_only'}
VAR_GLOBAL
    (* 生产就绪总状态；真实硬件全部人工映射并验证前必须为假。 *)
    bProductionReady : BOOL := FALSE;
    (* 当前操作模式。 *)
    eOperationMode : E_OperationMode;
    (* 当前控制源。 *)
    eControlSource : E_ControlSource;
    (* 当前机器状态。 *)
    eMachineState : E_MachineState;
    (* 当前初始化状态。 *)
    eInitializeState : E_InitializeState;
    (* 当前维护状态。 *)
    eMaintenanceState : E_MaintenanceState;
    (* 硬件绑定完成状态。 *)
    stHardwareBinding : ST_HardwareBindingStatus;
    (* 快速任务状态快照。 *)
    stFast : ST_FastStatus;
    (* 机器人接口状态。 *)
    stRobot : ST_RobotStatus;
    (* 供料器输入状态。 *)
    stFeeder : ST_FeederInput;
END_VAR

// ---- GVLs/GVL_Process.TcGVL
{attribute 'qualified_only'}
VAR_GLOBAL
    (* 当前快速过程实际值。 *)
    stActual : ST_ProcessActual;
    (* 当前周期提取特征。 *)
    stFeatures : ST_ProcessFeatures;
    (* 四个工艺步骤的判据结果。 *)
    astStepCriterion : ARRAY[1..4] OF ST_StepCriterionResult;
    (* 最近完成的周期结果。 *)
    stLastCycleResult : ST_CycleResult;
END_VAR

// ---- GVLs/GVL_Alarm.TcGVL
{attribute 'qualified_only'}
VAR_GLOBAL
    (* 各功能块发布的报警请求槽。 *)
    astRequests : ARRAY[1..64] OF ST_AlarmRequest;
    (* 汇总后的报警状态。 *)
    stStatus : ST_AlarmStatus;
    (* 报警确认命令请求编号。 *)
    nAcknowledgeRequestId : UDINT;
END_VAR

// ---- GVLs/GVL_Trace.TcGVL
{attribute 'qualified_only'}
VAR_GLOBAL
    (* 快速曲线环形缓冲区。 *)
    astCurveBuffer : ARRAY[0..2047] OF ST_CurveSample;
    (* 下一个曲线样本写入索引。 *)
    nWriteIndex : UINT;
    (* 当前曲线样本数量。 *)
    nSampleCount : UDINT;
    (* 曲线缓冲区是否发生覆盖。 *)
    bWrapped : BOOL;
END_VAR

// ---- GVLs/GVL_Persistent.TcGVL
{attribute 'qualified_only'}
VAR_GLOBAL PERSISTENT RETAIN
    (* 下一个焊接结果编号。 *)
    nNextWeldId : ULINT := 1;
    (* 持久化数据架构修订号。 *)
    nSchemaRevision : UDINT := 1;
    (* 最近激活的加工程序编号。 *)
    nLastActiveProgramId : UDINT;
END_VAR

// ---- GVLs/GVL_FastInternal.TcGVL
{attribute 'qualified_only'}
VAR_GLOBAL
    (* FastInputs按RequestId合同接受的完整快速命令快照。 *)
    stAcceptedCommand : ST_FastCommand;
END_VAR

// ---- POUs/Fast/PRG_FastInputs.TcPOU
PROGRAM PRG_FastInputs
VAR
    (* ---------------------------------------------------------
       四个力信号通道的一阶滤波实例数组。
       所属任务：Task_CffFast。
       唯一Owner：PRG_FastInputs。
       输入：同一EP3174工程力与四组时间常数。
       输出：ForceRaw、ForceCriterion、ForceControl、ForceDisplay。
       复位：硬件未映射、标定无效或处理参数无效时复位。
       --------------------------------------------------------- *)
    aFbForceChannelFilter : ARRAY[1..4] OF FB_LowPassFilter;
    (* ---------------------------------------------------------
       力测量链有效性实例。
       所属任务：Task_CffFast；唯一Owner：PRG_FastInputs。
       输入：EP3174诊断、映射状态、标定和工程力范围。
       输出：正式力有效位；Reset：链路未配置时复位。
       --------------------------------------------------------- *)
    fbForceSignalValidity : FB_SignalValidity;
    (* ---------------------------------------------------------
       外部位移一阶滤波实例。
       所属任务：Task_CffFast；唯一Owner：PRG_FastInputs。
       输入：经标定外部位移；输出：工艺位移绝对值。
       Reset：硬件未映射、标定或处理参数无效时复位。
       --------------------------------------------------------- *)
    fbDisplacementFilter : FB_LowPassFilter;
    (* ---------------------------------------------------------
       外部位移有效性实例。
       所属任务：Task_CffFast；唯一Owner：PRG_FastInputs。
       输入：位移诊断、映射、标定和范围；输出：正式有效位。
       Reset：位移链路未配置时复位。
       --------------------------------------------------------- *)
    fbDisplacementSignalValidity : FB_SignalValidity;
    (* ---------------------------------------------------------
       Collision Reference Sensor输入去抖实例。
       所属任务：Task_CffFast；唯一Owner：PRG_FastInputs。
       输入：未绑定数字输入占位；输出：稳定诊断状态。
       Reset：Collision输入未人工映射时复位。
       --------------------------------------------------------- *)
    fbCollisionDebounce : FB_Debounce;

    (* 实际快速任务配置周期，单位秒。 *)
    rCycleTime_s : LREAL;
    (* EP3174通道诊断是否无错误、无上溢且无下溢。 *)
    bForceDiagnosticOk : BOOL;
    (* 力标定结构是否通过基础版本、增益和方向检查。 *)
    bForceCalibrationValid : BOOL;
    (* 力测量链是否具备处理条件；未人工映射时保持FALSE。 *)
    bForcePathConfigured : BOOL;
    (* 经标定但尚未滤波的工程力，单位牛顿。 *)
    rConvertedForceN : LREAL;
    (* 位移输入诊断是否无错误、无上溢且无下溢。 *)
    bDisplacementDiagnosticOk : BOOL;
    (* 位移标定结构是否通过基础版本、增益和方向检查。 *)
    bDisplacementCalibrationValid : BOOL;
    (* 位移测量链是否具备处理条件；未人工映射时保持FALSE。 *)
    bDisplacementPathConfigured : BOOL;
    (* 经标定但尚未滤波的外部位移，单位毫米。 *)
    rConvertedDisplacementMm : LREAL;
    (* Collision标定结构是否有效。 *)
    bCollisionCalibrationValid : BOOL;
    (* Z轴真实驱动与轴状态是否允许使用NC位置诊断。 *)
    bAxisPositionValid : BOOL;
    (* Stable candidate used for the Main-to-Fast double-read acceptance. *)
    stFastCommandCandidate : ST_FastCommand;
    (* Live outer request identity sampled before copying the complete payload. *)
    udiLiveFastRequestId : UDINT;
END_VAR

(* ---------------------------------------------------------
   快速输入处理状态。
   目的：把未绑定过程映像占位转换为四路Force、外部位移、
         累计S_rel和Collision诊断契约。
   进入条件：每个Task_CffFast扫描调用。
   周期动作：检查映射/标定/诊断，滤波并发布类型化状态。
   正常出口：仅在用户完成映射且全部有效条件成立时发布有效位。
   超时：由各SignalValidity和Debounce实例按配置处理。
   NOK/Fault：任何输入无效即撤销对应有效位，不生成替代假值。
   --------------------------------------------------------- *)
(* Accept only a genuinely newer and stable complete Main-to-Fast package. *)
udiLiveFastRequestId := GVL_Command.stFast.nRequestId;
IF FC_IsNewerRequestId(
        udiCandidate := udiLiveFastRequestId,
        udiReference := GVL_FastInternal.stAcceptedCommand.nRequestId) THEN
    stFastCommandCandidate := GVL_Command.stFast;
    IF (stFastCommandCandidate.nRequestId = udiLiveFastRequestId)
        AND (GVL_Command.stFast.nRequestId = udiLiveFastRequestId) THEN
        GVL_FastInternal.stAcceptedCommand := stFastCommandCandidate;
    END_IF
END_IF

rCycleTime_s := UDINT_TO_LREAL(GVL_Config.stMachine.nFastTaskCycleUs) * 0.000001;

(* 力测量链：EP3174诊断、人工映射和受控标定必须同时有效。 *)
bForceDiagnosticOk := NOT GVL_IO.bForceChannelError
    AND NOT GVL_IO.bForceChannelOverrange
    AND NOT GVL_IO.bForceChannelUnderrange;
bForceCalibrationValid := FC_ValidateCalibration(
    bCalibrationValid := GVL_Calibration.stForce.bValid,
    udiRevision := GVL_Calibration.stForce.nRevision,
    rGain := GVL_Calibration.stForce.fGain,
    nDirection := GVL_Calibration.stForce.nDirection);
bForcePathConfigured := GVL_Status.stHardwareBinding.bForceInputMapped
    AND GVL_Config.stSensorProcessing.bValid
    AND bForceCalibrationValid;

IF bForceCalibrationValid THEN
    rConvertedForceN := ((INT_TO_LREAL(GVL_IO.nForceChannelRaw) - GVL_Calibration.stForce.fRawZero)
        * GVL_Calibration.stForce.fGain + GVL_Calibration.stForce.fOffsetN)
        * DINT_TO_LREAL(GVL_Calibration.stForce.nDirection);
ELSE
    rConvertedForceN := 0.0;
END_IF

fbForceSignalValidity(
    bEnable := GVL_Config.stSensorProcessing.bValid,
    bReset := NOT bForcePathConfigured,
    bRawValid := bForcePathConfigured AND bForceDiagnosticOk,
    rValue := rConvertedForceN,
    rMinimum := GVL_Config.stSensorProcessing.rForceMinimumN,
    rMaximum := GVL_Config.stSensorProcessing.rForceMaximumN,
    tInvalidDelay := GVL_Config.stSensorProcessing.tForceInvalidDelay);

(* 四个信号来自同一实际力，只允许滤波带宽不同，禁止ForceDisplay参与控制。 *)
aFbForceChannelFilter[1](bEnable := bForcePathConfigured, bReset := NOT bForcePathConfigured,
    bInputValid := fbForceSignalValidity.bValid, rInput := rConvertedForceN,
    rCycleTime_s := rCycleTime_s,
    rTimeConstant_s := GVL_Config.stSensorProcessing.arForceFilterTimeConstants_s[1]);
aFbForceChannelFilter[2](bEnable := bForcePathConfigured, bReset := NOT bForcePathConfigured,
    bInputValid := fbForceSignalValidity.bValid, rInput := rConvertedForceN,
    rCycleTime_s := rCycleTime_s,
    rTimeConstant_s := GVL_Config.stSensorProcessing.arForceFilterTimeConstants_s[2]);
aFbForceChannelFilter[3](bEnable := bForcePathConfigured, bReset := NOT bForcePathConfigured,
    bInputValid := fbForceSignalValidity.bValid, rInput := rConvertedForceN,
    rCycleTime_s := rCycleTime_s,
    rTimeConstant_s := GVL_Config.stSensorProcessing.arForceFilterTimeConstants_s[3]);
aFbForceChannelFilter[4](bEnable := bForcePathConfigured, bReset := NOT bForcePathConfigured,
    bInputValid := fbForceSignalValidity.bValid, rInput := rConvertedForceN,
    rCycleTime_s := rCycleTime_s,
    rTimeConstant_s := GVL_Config.stSensorProcessing.arForceFilterTimeConstants_s[4]);

GVL_Process.stActual.fForceRawN := aFbForceChannelFilter[1].rOutput;
GVL_Process.stActual.fForceCriterionN := aFbForceChannelFilter[2].rOutput;
GVL_Process.stActual.fForceControlN := aFbForceChannelFilter[3].rOutput;
GVL_Process.stActual.fForceDisplayN := aFbForceChannelFilter[4].rOutput;
GVL_Process.stActual.bForceValid := fbForceSignalValidity.bValid
    AND aFbForceChannelFilter[1].bValid AND aFbForceChannelFilter[2].bValid
    AND aFbForceChannelFilter[3].bValid AND aFbForceChannelFilter[4].bValid;

(* 外部位移链：该信号是正式SRelSensor主反馈，禁止自动降级为NC位置。 *)
bDisplacementDiagnosticOk := NOT GVL_IO.bDisplacementChannelError
    AND NOT GVL_IO.bDisplacementChannelOverrange
    AND NOT GVL_IO.bDisplacementChannelUnderrange;
bDisplacementCalibrationValid := FC_ValidateCalibration(
    bCalibrationValid := GVL_Calibration.stDisplacement.bValid,
    udiRevision := GVL_Calibration.stDisplacement.nRevision,
    rGain := GVL_Calibration.stDisplacement.fGainMmPerCount,
    nDirection := GVL_Calibration.stDisplacement.nDirection);
bDisplacementPathConfigured := GVL_Status.stHardwareBinding.bDisplacementInputMapped
    AND GVL_Config.stSensorProcessing.bValid
    AND bDisplacementCalibrationValid;

IF bDisplacementCalibrationValid THEN
    rConvertedDisplacementMm := ((INT_TO_LREAL(GVL_IO.nDisplacementChannelRaw)
        - GVL_Calibration.stDisplacement.fRawZero)
        * GVL_Calibration.stDisplacement.fGainMmPerCount
        + GVL_Calibration.stDisplacement.fOffsetMm)
        * DINT_TO_LREAL(GVL_Calibration.stDisplacement.nDirection);
ELSE
    rConvertedDisplacementMm := 0.0;
END_IF

fbDisplacementSignalValidity(
    bEnable := GVL_Config.stSensorProcessing.bValid,
    bReset := NOT bDisplacementPathConfigured,
    bRawValid := bDisplacementPathConfigured AND bDisplacementDiagnosticOk,
    rValue := rConvertedDisplacementMm,
    rMinimum := GVL_Config.stSensorProcessing.rDisplacementMinimumMm,
    rMaximum := GVL_Config.stSensorProcessing.rDisplacementMaximumMm,
    tInvalidDelay := GVL_Config.stSensorProcessing.tDisplacementInvalidDelay);
fbDisplacementFilter(
    bEnable := bDisplacementPathConfigured,
    bReset := NOT bDisplacementPathConfigured,
    bInputValid := fbDisplacementSignalValidity.bValid,
    rInput := rConvertedDisplacementMm,
    rCycleTime_s := rCycleTime_s,
    rTimeConstant_s := GVL_Config.stSensorProcessing.rDisplacementTimeConstant_s);

GVL_Process.stActual.fExternalDisplacementMm := fbDisplacementFilter.rOutput;
GVL_Process.stActual.bDisplacementValid := fbDisplacementSignalValidity.bValid
    AND fbDisplacementFilter.bValid;

(* Collision链同时要求人工数字输入映射、标定和真实轴位置有效。 *)
bCollisionCalibrationValid := GVL_Calibration.stCollision.bValid
    AND (GVL_Calibration.stCollision.nRevision > 0)
    AND (GVL_Calibration.stCollision.nSampleCount >= 3)
    AND FC_IsFiniteLReal(rValue := GVL_Calibration.stCollision.fReferencePositionMm);
bAxisPositionValid := GVL_Status.stHardwareBinding.bZAxisDriveLinked
    AND GVL_Status.stFast.stZAxis.bReady
    AND NOT GVL_Status.stFast.stZAxis.bError
    AND FC_IsFiniteLReal(rValue := GVL_Status.stFast.stZAxis.rActualPosition_mm);
fbCollisionDebounce(
    bEnable := GVL_Status.stHardwareBinding.bCollisionInputMapped,
    bReset := NOT GVL_Status.stHardwareBinding.bCollisionInputMapped,
    bInput := GVL_IO.bCollisionReferenceSensor,
    tOnDelay := GVL_Config.stSensorProcessing.tCollisionDebounce,
    tOffDelay := GVL_Config.stSensorProcessing.tCollisionDebounce);
GVL_Process.stActual.bCollisionSensorActive := fbCollisionDebounce.bOutput;
GVL_Process.stActual.bCollisionValid := GVL_Status.stHardwareBinding.bCollisionInputMapped
    AND bCollisionCalibrationValid AND bAxisPositionValid AND fbCollisionDebounce.bValid;

IF bCollisionCalibrationValid AND bAxisPositionValid THEN
    GVL_Process.stActual.fCollisionDeltaMm := GVL_Status.stFast.stZAxis.rActualPosition_mm
        - GVL_Calibration.stCollision.fReferencePositionMm;
ELSE
    GVL_Process.stActual.fCollisionDeltaMm := 0.0;
END_IF
GVL_Process.stActual.fCollisionReferenceMm := GVL_Process.stActual.fCollisionDeltaMm;

(* Contact参考点只按变化的RequestId处理一次，步骤切换绝不重置S_rel。 *)
IF GVL_Command.stProcessReference.udiContactReferenceRequestId
    <> GVL_Process.stActual.udiContactReferenceAcceptedId THEN
    GVL_Process.stActual.udiContactReferenceAcceptedId :=
        GVL_Command.stProcessReference.udiContactReferenceRequestId;

    IF GVL_Command.stProcessReference.bResetContactReference THEN
        GVL_Process.stActual.bContactReferenceValid := FALSE;
        GVL_Process.stActual.fContactSensorPositionMm := 0.0;
        GVL_Process.stActual.fContactAxisPositionMm := 0.0;
    ELSIF GVL_Command.stProcessReference.bLatchContactReference THEN
        IF GVL_Process.stActual.bForceValid AND GVL_Process.stActual.bDisplacementValid
            AND bAxisPositionValid THEN
            IF GVL_Command.stProcessReference.bUseProvidedContactReference THEN
                IF FC_IsFiniteLReal(rValue :=
                        GVL_Command.stProcessReference.rProvidedContactSensorPosition_mm)
                    AND FC_IsFiniteLReal(rValue :=
                        GVL_Command.stProcessReference.rProvidedContactAxisPosition_mm)
                    AND (GVL_Command.stProcessReference.rProvidedContactSensorPosition_mm
                        >= GVL_Config.stSensorProcessing.rDisplacementMinimumMm)
                    AND (GVL_Command.stProcessReference.rProvidedContactSensorPosition_mm
                        <= GVL_Config.stSensorProcessing.rDisplacementMaximumMm)
                    AND (GVL_Command.stProcessReference.rProvidedContactAxisPosition_mm
                        >= GVL_Config.stLimits.fZMinPositionMm)
                    AND (GVL_Command.stProcessReference.rProvidedContactAxisPosition_mm
                        <= GVL_Config.stLimits.fZMaxPositionMm) THEN
                    GVL_Process.stActual.fContactSensorPositionMm := GVL_Command.stProcessReference.rProvidedContactSensorPosition_mm;
                    GVL_Process.stActual.fContactAxisPositionMm := GVL_Command.stProcessReference.rProvidedContactAxisPosition_mm;
                    GVL_Process.stActual.bContactReferenceValid := TRUE;
                ELSE
                    GVL_Process.stActual.bContactReferenceValid := FALSE;
                    GVL_Process.stActual.fContactSensorPositionMm := 0.0;
                    GVL_Process.stActual.fContactAxisPositionMm := 0.0;
                END_IF
            ELSE
                GVL_Process.stActual.fContactSensorPositionMm := GVL_Process.stActual.fExternalDisplacementMm;
                GVL_Process.stActual.fContactAxisPositionMm := GVL_Status.stFast.stZAxis.rActualPosition_mm;
                GVL_Process.stActual.bContactReferenceValid := TRUE;
            END_IF
        ELSE
            GVL_Process.stActual.bContactReferenceValid := FALSE;
            GVL_Process.stActual.fContactSensorPositionMm := 0.0;
            GVL_Process.stActual.fContactAxisPositionMm := 0.0;
        END_IF
    END_IF
END_IF

IF GVL_Process.stActual.bContactReferenceValid AND GVL_Process.stActual.bDisplacementValid THEN
    GVL_Process.stActual.fSRelSensorMm := GVL_Process.stActual.fExternalDisplacementMm
        - GVL_Process.stActual.fContactSensorPositionMm;
ELSE
    GVL_Process.stActual.fSRelSensorMm := 0.0;
END_IF

IF GVL_Process.stActual.bContactReferenceValid AND bAxisPositionValid THEN
    GVL_Process.stActual.fSRelAxisMm := GVL_Status.stFast.stZAxis.rActualPosition_mm
        - GVL_Process.stActual.fContactAxisPositionMm;
ELSE
    GVL_Process.stActual.fSRelAxisMm := 0.0;
END_IF

GVL_Process.stActual.fAxisSensorDeltaMm := GVL_Process.stActual.fSRelAxisMm
    - GVL_Process.stActual.fSRelSensorMm;
GVL_Process.stActual.fRelativeDistanceMm := GVL_Process.stActual.fSRelSensorMm;
GVL_Process.stActual.bAxisSensorAgreement := GVL_Process.stActual.bContactReferenceValid
    AND GVL_Process.stActual.bDisplacementValid AND bAxisPositionValid
    AND (ABS(GVL_Process.stActual.fAxisSensorDeltaMm)
        <= ABS(GVL_Config.stSensorProcessing.rAxisSensorDeltaMaximumMm));

GVL_Process.stActual.bValid := GVL_Process.stActual.bForceValid
    AND GVL_Process.stActual.bDisplacementValid
    AND GVL_Process.stActual.bCollisionValid
    AND GVL_Process.stActual.bContactReferenceValid
    AND GVL_Process.stActual.bAxisSensorAgreement;

(* 发布Fast快照；未完成硬件映射时上述有效位自然保持FALSE。 *)
GVL_Status.stFast.nCycleCounter := GVL_Status.stFast.nCycleCounter + 1;
GVL_Status.stFast.nActualPeriodUs := GVL_Config.stMachine.nFastTaskCycleUs;
GVL_Status.stFast.stProcess := GVL_Process.stActual;

END_PROGRAM

// ---- POUs/FunctionBlocks/Utility/FB_LowPassFilter.TcPOU
FUNCTION_BLOCK FB_LowPassFilter
VAR_INPUT
    (* 滤波器运行许可；FALSE时撤销有效状态。 *)
    bEnable : BOOL;
    (* 算法复位请求；复位时清除历史值。 *)
    bReset : BOOL;
    (* 当前输入值是否可用于控制计算。 *)
    bInputValid : BOOL;
    (* 当前原始输入值。 *)
    rInput : LREAL;
    (* 实际调用周期，单位秒。 *)
    rCycleTime_s : LREAL;
    (* 一阶滤波时间常数，单位秒；零表示直接跟随。 *)
    rTimeConstant_s : LREAL;
END_VAR
VAR_OUTPUT
    (* 当前滤波输出；输入无效时保持最后有效值。 *)
    rOutput : LREAL;
    (* 本周期输出可用时为TRUE。 *)
    bValid : BOOL;
    (* 已接收过至少一个有效样本时为TRUE。 *)
    bInitialized : BOOL;
END_VAR
VAR
    (* 离散一阶滤波系数，限制在零到一。 *)
    rAlpha : LREAL;
END_VAR

(* 复位优先级最高：清除历史，且不得发布有效控制值。 *)
IF bReset OR NOT bEnable THEN
    rOutput := 0.0;
    bValid := FALSE;
    bInitialized := FALSE;
    RETURN;
END_IF

IF NOT bInputValid OR NOT FC_IsFiniteLReal(rValue := rInput) THEN
    (* 传感器无效时保持最后有效输出，但有效位立即撤销。 *)
    bValid := FALSE;
    RETURN;
END_IF

IF NOT bInitialized THEN
    rOutput := rInput;
    bInitialized := TRUE;
    bValid := TRUE;
    RETURN;
END_IF

IF rCycleTime_s <= 0.0 THEN
    (* 非正周期无法形成确定离散滤波，保持输出并撤销有效位。 *)
    bValid := FALSE;
    RETURN;
END_IF

IF rTimeConstant_s <= 0.0 THEN
    rOutput := rInput;
ELSE
    rAlpha := rCycleTime_s / (rTimeConstant_s + rCycleTime_s);
    rAlpha := FC_ClampLReal(rValue := rAlpha, rMinimum := 0.0, rMaximum := 1.0);
    rOutput := rOutput + rAlpha * (rInput - rOutput);
END_IF
bValid := TRUE;

END_FUNCTION_BLOCK

// ---- POUs/Functions/FC_IsFiniteLReal.TcPOU
FUNCTION FC_IsFiniteLReal : BOOL
VAR_INPUT
    (* 待检查的双精度值。 *)
    rValue : LREAL;
END_VAR
VAR CONSTANT
    (* 工程计算允许的对称有限上界，远高于本机物理量范围。 *)
    c_rEngineeringFiniteLimit : LREAL := 1.0E+300;
END_VAR

(* NaN不等于自身；正负无穷也会超出工程有限上界。 *)
FC_IsFiniteLReal := (rValue = rValue)
    AND (rValue <= c_rEngineeringFiniteLimit)
    AND (rValue >= -c_rEngineeringFiniteLimit);

END_FUNCTION

// ---- POUs/Functions/FC_ClampLReal.TcPOU
FUNCTION FC_ClampLReal : LREAL
VAR_INPUT
    (* 待限制的双精度数值。 *)
    rValue : LREAL;
    (* 允许区间的第一个边界；函数会自动处理上下限传反。 *)
    rMinimum : LREAL;
    (* 允许区间的第二个边界；函数会自动处理上下限传反。 *)
    rMaximum : LREAL;
END_VAR
VAR
    (* 归一化后的下边界。 *)
    rLow : LREAL;
    (* 归一化后的上边界。 *)
    rHigh : LREAL;
END_VAR

(* 先归一化边界，防止配方上下限传反后失去硬限制。 *)
IF rMinimum <= rMaximum THEN
    rLow := rMinimum;
    rHigh := rMaximum;
ELSE
    rLow := rMaximum;
    rHigh := rMinimum;
END_IF

IF rValue < rLow THEN
    FC_ClampLReal := rLow;
ELSIF rValue > rHigh THEN
    FC_ClampLReal := rHigh;
ELSE
    FC_ClampLReal := rValue;
END_IF

END_FUNCTION

// ---- POUs/Functions/FC_ValidateCalibration.TcPOU
FUNCTION FC_ValidateCalibration : BOOL
VAR_INPUT
    (* 标定流程发布的有效状态。 *)
    bCalibrationValid : BOOL;
    (* 标定修订号；零表示尚未形成受控版本。 *)
    udiRevision : UDINT;
    (* 标定比例增益，必须为非零有限值。 *)
    rGain : LREAL;
    (* 工程方向，只允许正一或负一。 *)
    nDirection : DINT;
END_VAR

(* 同时验证流程状态、版本、有限增益和方向，禁止只靠单一BOOL放行。 *)
FC_ValidateCalibration := bCalibrationValid
    AND (udiRevision > 0)
    AND FC_IsFiniteLReal(rValue := rGain)
    AND (ABS(rGain) > 0.0)
    AND ((nDirection = 1) OR (nDirection = -1));

END_FUNCTION

// ---- POUs/Fast/PRG_CffSequence.TcPOU
PROGRAM PRG_CffSequence
VAR
    fbContactDetect : FB_ContactDetect;
    fbForceDecline : FB_ForceDeclineObserver;
    fbStepCriterion : FB_StepProceedingCriterion;
    stContactInput : ST_ContactDetectInput;
    stForceDeclineInput : ST_ForceDeclineInput;
    stStepCriterionInput : ST_StepCriterionInput;
    stClearedStepCriterionResult : ST_StepCriterionResult;
    stStepResultCandidate : ST_StepCriterionResult;
    abStepResultWritten : ARRAY[1..4] OF BOOL;
    bStepResultPublishRequested : BOOL;
    bStepResultNok : BOOL;
    nStepResultIndex : INT := 1;

    eState : E_CffState := CFF_IDLE;
    eNextState : E_CffState := CFF_IDLE;
    ePreviousState : E_CffState := CFF_IDLE;
    bStateEntry : BOOL;
    eStep : E_CffStep := CFF_STEP_NONE;
    eSubPhase : E_StepSubPhase := STEP_SUBPHASE_NONE;
    eEndCause : E_StepEndCause := STEP_END_NONE;
    eExitIntent : E_CffExitIntent := CFF_EXIT_NONE;

    udiLastObservedCommandId : UDINT;
    udiActiveStartCommandId : UDINT;
    bNewSequenceCommand : BOOL;
    bStartEvent : BOOL;
    bStopEvent : BOOL;
    bAbortEvent : BOOL;
    bResetEvent : BOOL;
    nEventPulseCount : UINT;
    bStopRequestedLatched : BOOL;
    bResetPendingLatched : BOOL;
    bCycleNokLatched : BOOL;
    udiFirstFaultId : UDINT;
    stActiveSequenceCommand : ST_CffSequenceCommand;
    udiActiveCycleSnapshotRevision : UDINT;
    udiStartCycleSnapshotRevisionBefore : UDINT;
    udiStartMachineRevisionBefore : UDINT;
    udiStartForceProfileIdBefore : UDINT;
    udiStartForceProfileRevisionBefore : UDINT;
    udiStartRAxisProfileIdBefore : UDINT;
    udiStartRAxisProfileRevisionBefore : UDINT;
    bStartSourceSnapshotConsistent : BOOL;

    stCycleSnapshot : ST_CycleSnapshot;
    stMachineSnapshot : ST_MachineConfig;
    stLimitsSnapshot : ST_MachineLimits;
    stSequenceConfigSnapshot : ST_CffSequenceConfig;
    stZExtConfigSnapshot : ST_ZExtSetpointConfig;
    stForceProfileSnapshot : ST_ZForceControlProfile;
    stRAxisProfileSnapshot : ST_RAxisProfile;
    stFastConfigSnapshot : ST_CffFastConfigSnapshot;
    rCycleStartZPosition_mm : LREAL;
    rHardMaximumRelativePosition_mm : LREAL;
    rRequiredRelativePosition_mm : LREAL;
    rStepBoundary_mm : LREAL;
    rCycleTime_s : LREAL;
    nStepIndex : INT;

    stMotionIntent : ST_CffMotionIntent;
    udiZCommandId : UDINT;
    udiRCommandId : UDINT;
    stCandidateRCommand : ST_RAxisCommand;
    stLastPublishedRCommand : ST_RAxisCommand;
    bRCommandPayloadChanged : BOOL;

    stPendingProcessReferenceCommand : ST_ProcessReferenceCommand;
    udiContactReferenceRequestId : UDINT;
    udiExpectedContactReferenceAckId : UDINT;
    bProcessReferencePending : BOOL;
    bProcessReferenceResetPending : BOOL;
    bProcessReferenceLatchPending : BOOL;
    bApproachFaultStopPending : BOOL;
    bUnknownExternalRStopPending : BOOL;
    bSafeExitRStopPending : BOOL;
    bTerminalFaultStopRequired : BOOL;
    bUnloadTransferInitialized : BOOL;

    bBusy : BOOL;
    bDone : BOOL;
    bError : BOOL;
    bAborted : BOOL;
    bForceControlEnable : BOOL;
    bForceProfileTransfer : BOOL;
    bForceProfileTransferPending : BOOL;
    rForceTransferVelocity_mm_s : LREAL;
    rForceSet_kN : LREAL;
    rForceRamp_kN_s : LREAL;
    rSpeedSet_rpm : LREAL;
    rTargetRelativePosition_mm : LREAL;
    rStepTime_s : LREAL;
    rQualifiedForceHoldTime_s : LREAL;
    bRpmStopped : BOOL;
    bForceInBand : BOOL;
    nActiveStepProgramIndex : INT := 1;
    bStepTimingActive : BOOL;
    bStep4ProcessActive : BOOL;
    uliCycleDelta_us : ULINT;
    uliStepElapsed_us : ULINT;
    uliStepMaximum_us : ULINT;
    uliQualifiedHold_us : ULINT;
    uliQualifiedHoldTarget_us : ULINT;

    bPermissionValid : BOOL;
    bSnapshotIdentityValid : BOOL;
    bProgramValid : BOOL;
    bSequenceConfigValid : BOOL;
    bProfileValid : BOOL;
    bHardwareReady : BOOL;
    bSensorReady : BOOL;
    bExternalReady : BOOL;
    bLocalReturnTargetValid : BOOL;
    bHardForceActive : BOOL;
    bHardStrokeActive : BOOL;
    bCollisionLimitActive : BOOL;
    bExternalError : BOOL;
    bAxisError : BOOL;
    bSensorInvalid : BOOL;
    bPostContactSensorRequired : BOOL;
    bContactAcceptExactAck : BOOL;
    bContactAcceptInvalidReference : BOOL;
    bExternalProcessState : BOOL;
    bExternalOwnerHold : BOOL;
    bEntryMotionPermitted : BOOL;
    bSafeExitRequested : BOOL;
    bPrecheckExitRequested : BOOL;
    bSafeTerminalReset : BOOL;
    bUnloadHealthy : BOOL;
    bUnloadStandstillQualified : BOOL;
    bApproachNormalCompletion : BOOL;
    bReturnLevelHealthy : BOOL;
    bReturnEntryAuthorized : BOOL;
    bReturnPublicationAllowed : BOOL;
    bReturnSafeStopRequested : BOOL;
    bReturnEntryBlocked : BOOL;
    bEvaluateNok : BOOL;
    bEvaluateFault : BOOL;
    bStepResultHole : BOOL;
    bMissingStepResult : BOOL;
    nWrittenStepPrefix : INT;
    bContactResetPulse : BOOL;
    bForceDeclineResetPulse : BOOL;
    bStepCriterionResetPulse : BOOL;

    tonApproach : TON;
    tonRAxisStop : TON;
    tonStep4RAxisStop : TON;
    tonContactSearch : TON;
    tonContactReferenceAck : TON;
    tonControlledUnload : TON;
    tonUnloadStandstillConfirm : TON;
    tonExitRAxisStop : TON;
    tonReturn : TON;
END_VAR

(* Task_CffFast 中 CFF 流程、事务和安全状态机的唯一Owner：PRG_CffSequence。 *)
(* Scan pulses and scan-local defaults.  Transaction IDs and payloads are not reset. *)
bStartEvent := FALSE;
bStopEvent := FALSE;
bAbortEvent := FALSE;
bResetEvent := FALSE;
bForceProfileTransfer := FALSE;
bContactResetPulse := FALSE;
bForceDeclineResetPulse := FALSE;
bStepCriterionResetPulse := FALSE;
bStepResultPublishRequested := FALSE;
bStepResultNok := FALSE;
nStepResultIndex := 1;
eNextState := eState;
(* Every scan starts from an explicit no-motion level intent.  Active states below
   rebuild the complete package while source IDs remain monotonic and latched. *)
stMotionIntent.stZCommand.bEnable := FALSE;
stMotionIntent.stZCommand.bReset := FALSE;
stMotionIntent.stZCommand.bStop := FALSE;
stMotionIntent.stZCommand.bHome := FALSE;
stMotionIntent.stZCommand.bMoveAbsolute := FALSE;
stMotionIntent.stZCommand.bMoveVelocity := FALSE;
stMotionIntent.stZCommand.bUseExternalSetpoint := FALSE;
stMotionIntent.stZCommand.rHomePosition_mm := 0.0;
stMotionIntent.stZCommand.rPosition_mm := 0.0;
stMotionIntent.stZCommand.rVelocity_mm_s := 0.0;
stMotionIntent.stZCommand.rAcceleration_mm_s2 := 0.0;
stMotionIntent.stZCommand.rDeceleration_mm_s2 := 0.0;
stMotionIntent.stZCommand.eOwnerRequest := Z_OWNER_NONE;
stMotionIntent.bExternalEnableRequest := FALSE;
stMotionIntent.bExternalDisableRequest := FALSE;
stMotionIntent.rExternalTargetVelocity_mm_s := 0.0;
stMotionIntent.bRAxisProcessRequested := FALSE;
stMotionIntent.stRCommand.bEnable := TRUE;
stMotionIntent.stRCommand.bReset := FALSE;
stMotionIntent.stRCommand.bStop := TRUE;
stMotionIntent.stRCommand.bMoveVelocity := FALSE;
stMotionIntent.stRCommand.rVelocity_rpm := 0.0;
stMotionIntent.stRCommand.rAcceleration_rpm_s := stRAxisProfileSnapshot.fSpeedRampRpmS;
stMotionIntent.stRCommand.rDeceleration_rpm_s := stRAxisProfileSnapshot.fSpeedRampRpmS;
stMotionIntent.bForceProcessExitComplete := FALSE;
bForceControlEnable := FALSE;

(* One wrap-aware high-water mark covers every Sequence event type. *)
bNewSequenceCommand := FC_IsNewerRequestId(
    udiCandidate := GVL_FastInternal.stAcceptedCommand.stSequence.nCommandId,
    udiReference := udiLastObservedCommandId);
IF bNewSequenceCommand THEN
    nEventPulseCount := 0;
    IF GVL_FastInternal.stAcceptedCommand.stSequence.bStartPulse THEN
        nEventPulseCount := nEventPulseCount + 1;
    END_IF
    IF GVL_FastInternal.stAcceptedCommand.stSequence.bStopPulse THEN
        nEventPulseCount := nEventPulseCount + 1;
    END_IF
    IF GVL_FastInternal.stAcceptedCommand.stSequence.bAbortPulse THEN
        nEventPulseCount := nEventPulseCount + 1;
    END_IF
    IF GVL_FastInternal.stAcceptedCommand.stSequence.bResetPulse THEN
        nEventPulseCount := nEventPulseCount + 1;
    END_IF

    udiLastObservedCommandId := GVL_FastInternal.stAcceptedCommand.stSequence.nCommandId;
    IF nEventPulseCount > 1 THEN
        IF udiFirstFaultId = 0 THEN
            udiFirstFaultId := 16#0000A001;
        END_IF
    ELSE
        bStartEvent := GVL_FastInternal.stAcceptedCommand.stSequence.bStartPulse;
        bStopEvent := GVL_FastInternal.stAcceptedCommand.stSequence.bStopPulse;
        bAbortEvent := GVL_FastInternal.stAcceptedCommand.stSequence.bAbortPulse;
        bResetEvent := GVL_FastInternal.stAcceptedCommand.stSequence.bResetPulse;
    END_IF
END_IF

(* Safe terminal Reset is the only Reset allowed to clear algorithms and cycle state. *)
bSafeTerminalReset := (bResetEvent OR bResetPendingLatched)
    AND ((eState = CFF_IDLE) OR (eState = CFF_COMPLETE_OK) OR (eState = CFF_COMPLETE_NOK)
        OR (eState = CFF_ABORT) OR (eState = CFF_FAULT))
    AND NOT bBusy
    AND GVL_Status.stFast.stZAxis.bStandstill
    AND GVL_Status.stFast.stRAxis.bStandstill
    AND (GVL_Status.stFast.stZExtSetpoint.bReleaseOwner
        OR ((GVL_Status.stFast.stZExtSetpoint.eState = Z_EXT_IDLE)
            AND NOT GVL_Status.stFast.stZExtSetpoint.bEnabled));
IF bResetEvent AND NOT bSafeTerminalReset THEN
    bResetPendingLatched := TRUE;
    bStopRequestedLatched := TRUE;
    eExitIntent := CFF_EXIT_ABORT_NO_RETURN;
END_IF
IF bStopEvent OR bAbortEvent THEN
    bStopRequestedLatched := TRUE;
    eExitIntent := CFF_EXIT_ABORT_NO_RETURN;
END_IF

(* Frozen cycle validation is recomputed from the locally accepted Start snapshot. *)
bPermissionValid := stActiveSequenceCommand.bProductionPermission
    AND GVL_Command.stPermission.bAllowCycleStart
    AND GVL_Status.bProductionReady;
bSnapshotIdentityValid := (udiActiveStartCommandId > 0)
    AND bStartSourceSnapshotConsistent
    AND stCycleSnapshot.bValid
    AND (udiActiveCycleSnapshotRevision = stCycleSnapshot.nSnapshotRevision)
    AND (stActiveSequenceCommand.nProgramId
        = stCycleSnapshot.stProgram.stHeader.nProgramId)
    AND (stActiveSequenceCommand.nJoiningPointId
        = stCycleSnapshot.nJoiningPointId)
    AND (stCycleSnapshot.nMachineConfigRevision = stMachineSnapshot.nRevision)
    AND (stCycleSnapshot.nCalibrationRevision > 0)
    AND (stCycleSnapshot.nCalibrationRevision = GVL_Calibration.stForce.nRevision)
    AND (stCycleSnapshot.nCalibrationRevision = GVL_Calibration.stDisplacement.nRevision)
    AND (stCycleSnapshot.nCalibrationRevision = GVL_Calibration.stCollision.nRevision)
    AND (stCycleSnapshot.stProgram.stHeader.nToolId = stMachineSnapshot.nToolId)
    AND (stCycleSnapshot.stProgram.stHeader.nAnvilId = stMachineSnapshot.nAnvilId);
bProgramValid := FC_ValidateJoinProgram(
    stProgram := stCycleSnapshot.stProgram,
    stMachineLimits := stLimitsSnapshot);
bSequenceConfigValid := FC_ValidateCffSequenceConfig(
    stConfig := stSequenceConfigSnapshot,
    stLimits := stLimitsSnapshot);
bProfileValid := stForceProfileSnapshot.bValid
    AND (stForceProfileSnapshot.nProfileId > 0)
    AND (stForceProfileSnapshot.nRevision > 0)
    AND stRAxisProfileSnapshot.bValid
    AND (stRAxisProfileSnapshot.nProfileId > 0)
    AND (stRAxisProfileSnapshot.nRevision > 0)
    AND (stCycleSnapshot.stProgram.stHeader.nForceProfileId
        = stForceProfileSnapshot.nProfileId)
    AND (stCycleSnapshot.stProgram.stHeader.nRAxisProfileId
        = stRAxisProfileSnapshot.nProfileId)
    AND FC_IsFiniteLReal(rValue := stRAxisProfileSnapshot.fTargetSpeedRpm)
    AND FC_IsFiniteLReal(rValue := stRAxisProfileSnapshot.fSpeedRampRpmS)
    AND FC_IsFiniteLReal(rValue := stRAxisProfileSnapshot.fAccelerationTimeS)
    AND FC_IsFiniteLReal(rValue := stRAxisProfileSnapshot.fDecelerationTimeS)
    AND FC_IsFiniteLReal(rValue := stRAxisProfileSnapshot.fMinimumQualifiedSpeedRpm)
    AND (stRAxisProfileSnapshot.fSpeedRampRpmS > 0.0)
    AND (stRAxisProfileSnapshot.fAccelerationTimeS > 0.0)
    AND (stRAxisProfileSnapshot.fDecelerationTimeS > 0.0)
    AND (ABS(stRAxisProfileSnapshot.fTargetSpeedRpm) <= stLimitsSnapshot.fRMaxSpeedRpm)
    AND (stRAxisProfileSnapshot.fMinimumQualifiedSpeedRpm >= 0.0)
    AND (stRAxisProfileSnapshot.fMinimumQualifiedSpeedRpm <= stLimitsSnapshot.fRMaxSpeedRpm);
bHardwareReady := GVL_Status.stHardwareBinding.bZAxisNcAssigned
    AND GVL_Status.stHardwareBinding.bRAxisNcAssigned
    AND GVL_Status.stHardwareBinding.bZAxisDriveLinked
    AND GVL_Status.stHardwareBinding.bRAxisDriveLinked
    AND GVL_Status.stHardwareBinding.bForceInputMapped
    AND GVL_Status.stHardwareBinding.bDisplacementInputMapped
    AND GVL_Status.stHardwareBinding.bCollisionInputMapped
    AND GVL_Status.stHardwareBinding.bProductionHardwareBindingComplete
    AND GVL_Status.stFast.stZAxis.bReady
    AND GVL_Status.stFast.stZAxis.bHomed
    AND GVL_Status.stFast.stZAxis.bStandstill
    AND NOT GVL_Status.stFast.stZAxis.bError
    AND GVL_Status.stFast.stRAxis.bReady
    AND GVL_Status.stFast.stRAxis.bStandstill
    AND NOT GVL_Status.stFast.stRAxis.bError;
bExternalReady := GVL_Status.stFast.stZExtSetpoint.bReleaseOwner
    OR ((GVL_Status.stFast.stZExtSetpoint.eState = Z_EXT_IDLE)
        AND NOT GVL_Status.stFast.stZExtSetpoint.bEnabled);
bLocalReturnTargetValid := FC_IsFiniteLReal(rValue := rCycleStartZPosition_mm)
    AND rCycleStartZPosition_mm >= stLimitsSnapshot.fZMinPositionMm
    AND rCycleStartZPosition_mm <= stLimitsSnapshot.fZMaxPositionMm;

(* Compute current-scan safety facts before any algorithm consumes them. *)
bPostContactSensorRequired := (eState >= CFF_STEP1_ENTRY)
    AND (eState <= CFF_EXTSETPOINT_DISABLE);
bHardForceActive := bBusy
    AND GVL_Process.stActual.bForceValid
    AND FC_IsFiniteLReal(rValue := GVL_Process.stActual.fForceControlN)
    AND (GVL_Process.stActual.fForceControlN >= stLimitsSnapshot.fMaxForceN);
bHardStrokeActive := bBusy
    AND bPostContactSensorRequired
    AND GVL_Process.stActual.bContactReferenceValid
    AND FC_IsFiniteLReal(rValue := GVL_Process.stActual.fSRelSensorMm)
    AND FC_IsFiniteLReal(rValue := rHardMaximumRelativePosition_mm)
    AND (GVL_Process.stActual.fSRelSensorMm >= rHardMaximumRelativePosition_mm);
bCollisionLimitActive := bBusy AND GVL_Process.stActual.bCollisionValid
    AND GVL_Process.stActual.bCollisionSensorActive;
bSensorReady := GVL_Process.stActual.bForceValid
    AND GVL_Process.stActual.bDisplacementValid
    AND GVL_Process.stActual.bCollisionValid
    AND NOT bHardForceActive
    AND NOT bHardStrokeActive
    AND NOT bCollisionLimitActive;
bExternalError := GVL_Status.stFast.stZExtSetpoint.bError
    OR GVL_Status.stFast.stZExternalTrajectory.bFault;
bAxisError := GVL_Status.stFast.stZAxis.bError OR GVL_Status.stFast.stRAxis.bError;
bContactAcceptExactAck := (eState = CFF_CONTACT_ACCEPT)
    AND bProcessReferenceLatchPending
    AND (GVL_Process.stActual.udiContactReferenceAcceptedId
        = udiExpectedContactReferenceAckId);
bContactAcceptInvalidReference := bContactAcceptExactAck
    AND NOT GVL_Process.stActual.bContactReferenceValid;
bSensorInvalid := bBusy AND NOT bContactAcceptInvalidReference
    AND (NOT GVL_Process.stActual.bForceValid
    OR NOT GVL_Process.stActual.bDisplacementValid
    OR NOT GVL_Process.stActual.bCollisionValid
    OR NOT FC_IsFiniteLReal(rValue := GVL_Process.stActual.fForceControlN)
    OR NOT FC_IsFiniteLReal(rValue := GVL_Process.stActual.fForceCriterionN)
    OR NOT FC_IsFiniteLReal(rValue := GVL_Process.stActual.fSRelSensorMm)
    OR NOT FC_IsFiniteLReal(rValue := GVL_Status.stFast.stRAxis.rActualVelocity_rpm)
    OR (bPostContactSensorRequired
        AND (NOT GVL_Process.stActual.bValid
            OR NOT GVL_Process.stActual.bContactReferenceValid
            OR NOT GVL_Process.stActual.bAxisSensorAgreement)));

IF bStartEvent AND bBusy THEN
    IF udiFirstFaultId = 0 THEN
        udiFirstFaultId := 16#0000A001;
    END_IF
END_IF
IF bBusy AND (udiActiveStartCommandId > 0)
    AND (eState <> CFF_IDLE)
    AND NOT bContactAcceptInvalidReference
    AND ((GVL_Calibration.stForce.nRevision <> stCycleSnapshot.nCalibrationRevision)
        OR (GVL_Calibration.stDisplacement.nRevision <> stCycleSnapshot.nCalibrationRevision)
        OR (GVL_Calibration.stCollision.nRevision <> stCycleSnapshot.nCalibrationRevision)) THEN
    IF udiFirstFaultId = 0 THEN
        udiFirstFaultId := 16#0000A00F;
    END_IF
END_IF

(* Deterministic first-cause mapping applies from Approach through every safe terminal. *)
IF (eState >= CFF_APPROACH)
    AND (eState <= CFF_FAULT) AND (udiFirstFaultId = 0) THEN
    IF bHardForceActive THEN
        udiFirstFaultId := 16#0000A00C;
    ELSIF bHardStrokeActive THEN
        udiFirstFaultId := 16#0000A00D;
    ELSIF bCollisionLimitActive THEN
        udiFirstFaultId := 16#0000A00E;
    ELSIF (eState = CFF_CONTROLLED_FORCE_UNLOAD)
        AND (GVL_Status.stFast.stZForceControl.bFault
            OR NOT GVL_Status.stFast.stZForceControl.bActive
            OR NOT GVL_Status.stFast.bForceSetpointRampValid
            OR NOT FC_IsFiniteLReal(rValue := rForceRamp_kN_s)
            OR (rForceRamp_kN_s <= 0.0)) THEN
        udiFirstFaultId := 16#0000A00B;
    ELSIF bSensorInvalid THEN
        udiFirstFaultId := 16#0000A00F;
    ELSIF GVL_Status.stFast.stZAxis.bError THEN
        udiFirstFaultId := 16#0000A010;
    ELSIF GVL_Status.stFast.stRAxis.bError THEN
        udiFirstFaultId := 16#0000A011;
    ELSIF bExternalError THEN
        udiFirstFaultId := 16#0000A012;
    END_IF
END_IF

bEntryMotionPermitted := NOT (bStopRequestedLatched OR bAbortEvent
    OR bResetPendingLatched OR bHardForceActive OR bHardStrokeActive
    OR bCollisionLimitActive OR bExternalError OR bAxisError OR bSensorInvalid
    OR (udiFirstFaultId > 0));
bReturnEntryBlocked := bStopRequestedLatched OR bAbortEvent
    OR bResetPendingLatched OR bHardForceActive OR bHardStrokeActive
    OR bCollisionLimitActive OR bExternalError OR bAxisError OR bSensorInvalid
    OR (udiFirstFaultId > 0);
bApproachNormalCompletion := NOT bStateEntry
    AND (GVL_Status.stFast.udiAcceptedSequenceZCommandId = udiZCommandId)
    AND GVL_Status.stFast.stZAxis.bDone
    AND GVL_Status.stFast.stZAxis.bStandstill
    AND (GVL_Status.stFast.udiAcceptedSequenceRCommandId = udiRCommandId)
    AND GVL_Status.stFast.stRAxis.bStandstill;
bReturnLevelHealthy := GVL_Status.stFast.stZExtSetpoint.bReleaseOwner
    AND (GVL_Status.stFast.udiAcceptedSequenceRCommandId = udiRCommandId)
    AND GVL_Status.stFast.stRAxis.bStandstill
    AND GVL_Status.stFast.stZAxis.bReady
    AND GVL_Status.stFast.stRAxis.bReady
    AND NOT GVL_Status.stFast.stZAxis.bError
    AND NOT GVL_Status.stFast.stRAxis.bError
    AND NOT GVL_Status.stFast.stZExtSetpoint.bError
    AND NOT GVL_Status.stFast.stZExternalTrajectory.bFault;
bReturnEntryAuthorized := bReturnLevelHealthy
    AND GVL_Status.stFast.stZAxis.bStandstill;
bReturnPublicationAllowed := NOT bReturnEntryBlocked
    AND bReturnLevelHealthy
    AND (NOT bStateEntry OR bReturnEntryAuthorized);

bPrecheckExitRequested := bStopRequestedLatched OR bAbortEvent
    OR bResetPendingLatched OR (udiFirstFaultId > 0);

(* 受控卸载必须建立在已接管的Force与External生命周期上，原始传感器布尔值不能单独启用PI。 *)
bUnloadHealthy := GVL_Process.stActual.bForceValid
    AND GVL_Process.stActual.bContactReferenceValid
    AND GVL_Process.stActual.bAxisSensorAgreement
    AND GVL_Status.stFast.bForceSetpointRampValid
    AND GVL_Status.stFast.stZForceControl.bActive
    AND FC_IsFiniteLReal(rValue := rForceRamp_kN_s)
    AND FC_IsFiniteLReal(rValue := GVL_Process.stActual.fForceControlN)
    AND FC_IsFiniteLReal(rValue := GVL_Process.stActual.fSRelSensorMm)
    AND rForceRamp_kN_s > 0
    AND GVL_Status.stFast.stZExtSetpoint.bEnabled
    AND GVL_Status.stFast.stZExtSetpoint.bAcceptedSetpointValid
    AND GVL_Status.stFast.stZExternalTrajectory.bActive
    AND FC_IsFiniteLReal(
        rValue := GVL_Status.stFast.stZExtSetpoint.rAcceptedVelocity_mm_s)
    AND NOT bExternalError
    AND NOT bAxisError
    AND NOT bSensorInvalid
    AND NOT GVL_Status.stFast.stZForceControl.bFault
    AND NOT GVL_Status.stFast.stZExternalTrajectory.bFault;
bUnloadStandstillQualified := GVL_Status.stFast.bForceSetpointRampValid
    AND GVL_Status.stFast.bForceSetpointRampReached
    AND ABS(GVL_Process.stActual.fForceControlN)
        <= stCycleSnapshot.stProgram.stHeader.fContactForceOffN
    AND ABS(GVL_Status.stFast.stZExtSetpoint.rAcceptedVelocity_mm_s)
        <= stZExtConfigSnapshot.rStandstillVelocity_mm_s
    AND bUnloadHealthy;

(* Step classification, Entry Reset and saturated clocks are resolved before
   either stateful algorithm is called.  The index always remains in 1..4. *)
nActiveStepProgramIndex := 1;
IF (eState = CFF_STEP2_ENTRY) OR (eState = CFF_STEP2_RAMP_PROCESS)
    OR (eState = CFF_STEP2_END_CHECK) THEN
    nActiveStepProgramIndex := 2;
ELSIF (eState = CFF_STEP3_ENTRY) OR (eState = CFF_STEP3_RAMP_PROCESS)
    OR (eState = CFF_STEP3_END_CHECK) THEN
    nActiveStepProgramIndex := 3;
ELSIF (eState = CFF_BRAKE_AND_COMPRESSION_RAMP)
    OR (eState = CFF_STEP4_VALID_FORCE_HOLD) THEN
    nActiveStepProgramIndex := 4;
END_IF

bForceDeclineResetPulse := bStateEntry
    AND ((eState = CFF_STEP1_ENTRY)
        OR (eState = CFF_STEP2_ENTRY)
        OR (eState = CFF_STEP3_ENTRY));
bStepCriterionResetPulse := bStateEntry
    AND ((eState = CFF_STEP1_ENTRY)
        OR (eState = CFF_STEP2_ENTRY)
        OR (eState = CFF_STEP3_ENTRY)
        OR (eState = CFF_BRAKE_AND_COMPRESSION_RAMP));

IF bStateEntry
    AND ((eState = CFF_STEP1_ENTRY)
        OR (eState = CFF_STEP2_ENTRY)
        OR (eState = CFF_STEP3_ENTRY)
        OR (eState = CFF_BRAKE_AND_COMPRESSION_RAMP)) THEN
    uliStepElapsed_us := 0;
END_IF
IF bStateEntry AND (eState = CFF_BRAKE_AND_COMPRESSION_RAMP) THEN
    uliQualifiedHold_us := 0;
END_IF

uliCycleDelta_us := UDINT_TO_ULINT(stMachineSnapshot.nFastTaskCycleUs);
uliStepMaximum_us :=
    UDINT_TO_ULINT(stCycleSnapshot.stProgram.astSteps[nActiveStepProgramIndex].stProceeding.nStepMaxMs)
    * ULINT#1000;
uliQualifiedHoldTarget_us :=
    UDINT_TO_ULINT(stCycleSnapshot.stProgram.astSteps[4].stProceeding.nQualifiedForceHoldMs)
    * ULINT#1000;
bStepTimingActive := (eState = CFF_STEP1_RAMP_PROCESS)
    OR (eState = CFF_STEP2_RAMP_PROCESS)
    OR (eState = CFF_STEP3_RAMP_PROCESS)
    OR (eState = CFF_BRAKE_AND_COMPRESSION_RAMP)
    OR (eState = CFF_STEP4_VALID_FORCE_HOLD);
bStep4ProcessActive := (eState = CFF_BRAKE_AND_COMPRESSION_RAMP)
    OR (eState = CFF_STEP4_VALID_FORCE_HOLD);
IF bStepTimingActive THEN
    IF uliStepElapsed_us < uliStepMaximum_us THEN
        IF uliCycleDelta_us >= uliStepMaximum_us - uliStepElapsed_us THEN
            uliStepElapsed_us := uliStepMaximum_us;
        ELSE
            uliStepElapsed_us := uliStepElapsed_us + uliCycleDelta_us;
        END_IF
    END_IF
END_IF
rStepTime_s := ULINT_TO_LREAL(uliStepElapsed_us) * 0.000001;

IF bStep4ProcessActive
    AND GVL_Process.stActual.bForceValid
    AND FC_IsFiniteLReal(rValue := GVL_Process.stActual.fForceControlN)
    AND FC_IsFiniteLReal(rValue := GVL_Status.stFast.stRAxis.rActualVelocity_rpm) THEN
    bRpmStopped := ABS(GVL_Status.stFast.stRAxis.rActualVelocity_rpm)
        <= stCycleSnapshot.stProgram.astSteps[4].stProceeding.fRpmStoppedThresholdRpm;
    bForceInBand := ABS(
        GVL_Process.stActual.fForceControlN
        - stCycleSnapshot.stProgram.astSteps[4].fSetForceN)
        <= stCycleSnapshot.stProgram.astSteps[4].stProceeding.fForceBandToleranceN;
    IF bRpmStopped AND bForceInBand THEN
        IF uliQualifiedHold_us < uliQualifiedHoldTarget_us THEN
            IF uliCycleDelta_us >= uliQualifiedHoldTarget_us - uliQualifiedHold_us THEN
                uliQualifiedHold_us := uliQualifiedHoldTarget_us;
            ELSE
                uliQualifiedHold_us := uliQualifiedHold_us + uliCycleDelta_us;
            END_IF
        END_IF
    END_IF
ELSE
    bRpmStopped := FALSE;
    bForceInBand := FALSE;
END_IF
rQualifiedForceHoldTime_s := ULINT_TO_LREAL(uliQualifiedHold_us) * 0.000001;

(* Algorithms use this scan's local state, never the previously published mirror. *)
rCycleTime_s := UDINT_TO_LREAL(stMachineSnapshot.nFastTaskCycleUs) * 0.000001;
stContactInput.bEnable := eState = CFF_CONTACT_SEARCH;
stContactInput.bReset := bSafeTerminalReset OR bContactResetPulse;
stContactInput.rForceActual_kN := GVL_Process.stActual.fForceCriterionN * 0.001;
stContactInput.rForceOn_kN := stCycleSnapshot.stProgram.stHeader.fContactForceOnN * 0.001;
stContactInput.rForceOff_kN := stCycleSnapshot.stProgram.stHeader.fContactForceOffN * 0.001;
stContactInput.rAxisPosition_mm := GVL_Status.stFast.stZAxis.rActualPosition_mm;
stContactInput.rSensorPosition_mm := GVL_Process.stActual.fExternalDisplacementMm;
stContactInput.rAxisPositionMinimum_mm := stLimitsSnapshot.fZMinPositionMm;
stContactInput.rAxisPositionMaximum_mm := stLimitsSnapshot.fZMaxPositionMm;
stContactInput.rSensorPositionMinimum_mm := stCycleSnapshot.stProgram.stHeader.fContactSensorMinimumMm;
stContactInput.rSensorPositionMaximum_mm := stCycleSnapshot.stProgram.stHeader.fContactSensorMaximumMm;
stContactInput.rAxisVelocity_mm_s := GVL_Status.stFast.stZAxis.rActualVelocity_mm_s;
stContactInput.rCaptureMaximumVelocity_mm_s := stCycleSnapshot.stProgram.stHeader.fContactSearchVelocityMmS;
stContactInput.rDebounceTime_s := UDINT_TO_LREAL(stCycleSnapshot.stProgram.stHeader.nContactDebounceMs) * 0.001;
stContactInput.rCycleTime_s := rCycleTime_s;
stContactInput.bSignalValid := GVL_Process.stActual.bForceValid
    AND GVL_Process.stActual.bDisplacementValid
    AND GVL_Status.stFast.stZAxis.bReady
    AND stCycleSnapshot.bValid;
fbContactDetect(stInput := stContactInput);

stForceDeclineInput.bEnable :=
    ((eState = CFF_STEP1_RAMP_PROCESS)
        OR (eState = CFF_STEP2_RAMP_PROCESS)
        OR (eState = CFF_STEP3_RAMP_PROCESS))
    AND (stCycleSnapshot.stProgram.astSteps[nActiveStepProgramIndex].stProceeding.ePrimaryCriterion
        = STEP_CRIT_FORCE_DECLINE_TO);
stForceDeclineInput.bReset := bSafeTerminalReset OR bForceDeclineResetPulse;
stForceDeclineInput.bSignalValid := GVL_Process.stActual.bForceValid
    AND GVL_Process.stActual.bDisplacementValid
    AND GVL_Process.stActual.bContactReferenceValid
    AND GVL_Process.stActual.bAxisSensorAgreement
    AND NOT bSensorInvalid
    AND NOT bAxisError
    AND NOT bExternalError;
stForceDeclineInput.rForceActual_kN := GVL_Process.stActual.fForceCriterionN * 0.001;
stForceDeclineInput.rSpeed_rpm := GVL_Status.stFast.stRAxis.rActualVelocity_rpm;
stForceDeclineInput.rRelativePosition_mm := GVL_Process.stActual.fSRelSensorMm;
stForceDeclineInput.rAxisVelocity_mm_s := GVL_Status.stFast.stZAxis.rActualVelocity_mm_s;
stForceDeclineInput.rStepTime_s := rStepTime_s;
stForceDeclineInput.rArmForce_kN :=
    stCycleSnapshot.stProgram.astSteps[nActiveStepProgramIndex].stProceeding.fArmForceN * 0.001;
stForceDeclineInput.rDeclineTo_kN :=
    stCycleSnapshot.stProgram.astSteps[nActiveStepProgramIndex].stProceeding.fDeclineToN * 0.001;
stForceDeclineInput.rHysteresis_kN :=
    stCycleSnapshot.stProgram.astSteps[nActiveStepProgramIndex].stProceeding.fDeclineHysteresisN * 0.001;
stForceDeclineInput.rMinimumDeclineRate_kN_s :=
    stCycleSnapshot.stProgram.astSteps[nActiveStepProgramIndex].stProceeding.fMinimumDeclineRateNS * 0.001;
stForceDeclineInput.rCriterionSRelMinimum_mm :=
    stCycleSnapshot.stProgram.astSteps[nActiveStepProgramIndex].stProceeding.fCriterionSRelMinMm;
stForceDeclineInput.rCriterionSRelMaximum_mm :=
    stCycleSnapshot.stProgram.astSteps[nActiveStepProgramIndex].stProceeding.fCriterionSRelMaxMm;
stForceDeclineInput.rCriterionRpmMinimum :=
    stCycleSnapshot.stProgram.astSteps[nActiveStepProgramIndex].stProceeding.fCriterionRpmMin;
stForceDeclineInput.rCaptureMaximumVelocity_mm_s :=
    stCycleSnapshot.stProgram.astSteps[nActiveStepProgramIndex].stProceeding.fCaptureMaxVelocityMmS;
stForceDeclineInput.rDebounceTime_s :=
    UDINT_TO_LREAL(stCycleSnapshot.stProgram.astSteps[nActiveStepProgramIndex].stProceeding.nDeclineDebounceMs)
    * 0.001;
stForceDeclineInput.rCycleTime_s := rCycleTime_s;
fbForceDecline(stInput := stForceDeclineInput);

stStepCriterionInput.bEnable := (eState = CFF_STEP1_RAMP_PROCESS)
    OR (eState = CFF_STEP2_RAMP_PROCESS)
    OR (eState = CFF_STEP3_RAMP_PROCESS)
    OR (eState = CFF_BRAKE_AND_COMPRESSION_RAMP)
    OR (eState = CFF_STEP4_VALID_FORCE_HOLD);
stStepCriterionInput.bReset := bSafeTerminalReset OR bStepCriterionResetPulse;
stStepCriterionInput.bSignalValid :=
    stCycleSnapshot.stProgram.astSteps[nActiveStepProgramIndex].stProceeding.bValid
    AND GVL_Process.stActual.bForceValid
    AND GVL_Process.stActual.bDisplacementValid
    AND GVL_Process.stActual.bCollisionValid
    AND GVL_Process.stActual.bContactReferenceValid
    AND GVL_Process.stActual.bAxisSensorAgreement
    AND NOT bSensorInvalid;
stStepCriterionInput.ePrimaryCriterion :=
    stCycleSnapshot.stProgram.astSteps[nActiveStepProgramIndex].stProceeding.ePrimaryCriterion;
stStepCriterionInput.eSecondaryAction :=
    stCycleSnapshot.stProgram.astSteps[nActiveStepProgramIndex].stProceeding.eSecondaryAction;
stStepCriterionInput.rRelativePosition_mm := GVL_Process.stActual.fSRelSensorMm;
stStepCriterionInput.rRelativeDistanceTarget_mm :=
    stCycleSnapshot.stProgram.astSteps[nActiveStepProgramIndex].stProceeding.fRelativeDistanceMm;
stStepCriterionInput.rStepTime_s := rStepTime_s;
stStepCriterionInput.rStepTimeTarget_s :=
    UDINT_TO_LREAL(stCycleSnapshot.stProgram.astSteps[nActiveStepProgramIndex].stProceeding.nPrimaryStepTimeMs)
    * 0.001;
stStepCriterionInput.rStepMinimumTime_s :=
    UDINT_TO_LREAL(stCycleSnapshot.stProgram.astSteps[nActiveStepProgramIndex].stProceeding.nStepMinMs)
    * 0.001;
stStepCriterionInput.rStepMaximumTime_s :=
    ULINT_TO_LREAL(uliStepMaximum_us) * 0.000001;
stStepCriterionInput.rForceActual_kN := GVL_Process.stActual.fForceCriterionN * 0.001;
stStepCriterionInput.bForceDeclineArmed := fbForceDecline.stOutput.bArmed;
stStepCriterionInput.bForceDeclineConfirmed := fbForceDecline.stOutput.bConfirmed;
stStepCriterionInput.rSecondaryDistanceLimit_mm :=
    stCycleSnapshot.stProgram.astSteps[nActiveStepProgramIndex].stProceeding.fSecondarySRelMm;
stStepCriterionInput.bHardForceActive := bHardForceActive;
stStepCriterionInput.bHardStrokeActive := bHardStrokeActive;
stStepCriterionInput.bCollisionActive := bCollisionLimitActive;
stStepCriterionInput.bSensorInvalid := bSensorInvalid;
stStepCriterionInput.bAxisFault := bAxisError OR bExternalError;
stStepCriterionInput.bStopRequested := bStopRequestedLatched;
fbStepCriterion(stInput := stStepCriterionInput);

(* Current algorithm/ramp faults become the first fault before event-priority
   routing.  Entry scans are excluded because their new targets are not yet ACKed. *)
IF bBusy AND (udiFirstFaultId = 0) THEN
    IF ((eState = CFF_STEP1_RAMP_PROCESS)
        OR (eState = CFF_STEP2_RAMP_PROCESS)
        OR (eState = CFF_STEP3_RAMP_PROCESS))
        AND (fbForceDecline.stOutput.bFault OR fbStepCriterion.stOutput.bFault) THEN
        udiFirstFaultId := 16#0000A00B;
    ELSIF (((eState = CFF_BRAKE_AND_COMPRESSION_RAMP) AND NOT bStateEntry)
        OR (eState = CFF_STEP4_VALID_FORCE_HOLD))
        AND (fbForceDecline.stOutput.bFault OR fbStepCriterion.stOutput.bFault
            OR NOT GVL_Status.stFast.bForceSetpointRampValid
            OR NOT GVL_Status.stFast.bRSpeedRampValid) THEN
        udiFirstFaultId := 16#0000A00B;
    END_IF
END_IF

(* Every timer is called once per scan, outside the state CASE. *)
tonApproach(
    IN := (eState = CFF_APPROACH) AND NOT bApproachNormalCompletion,
    PT := stSequenceConfigSnapshot.tApproachTimeout);
tonRAxisStop(
    IN := (eState = CFF_APPROACH)
        AND NOT ((GVL_Status.stFast.udiAcceptedSequenceRCommandId = udiRCommandId)
            AND GVL_Status.stFast.stRAxis.bStandstill),
    PT := stSequenceConfigSnapshot.tRAxisStopTimeout);
tonStep4RAxisStop(
    IN := ((eState = CFF_BRAKE_AND_COMPRESSION_RAMP)
            OR (eState = CFF_STEP4_VALID_FORCE_HOLD))
        AND ((eState = CFF_BRAKE_AND_COMPRESSION_RAMP AND bStateEntry)
            OR NOT ((GVL_Status.stFast.udiAcceptedSequenceRCommandId = udiRCommandId)
                AND bRpmStopped)),
    PT := stSequenceConfigSnapshot.tRAxisStopTimeout);
tonContactSearch(IN := eState = CFF_CONTACT_SEARCH, PT := stSequenceConfigSnapshot.tContactSearchTimeout);
tonContactReferenceAck(IN := bProcessReferencePending, PT := stSequenceConfigSnapshot.tContactReferenceAckTimeout);
tonControlledUnload(
    IN := eState = CFF_CONTROLLED_FORCE_UNLOAD,
    PT := stSequenceConfigSnapshot.tControlledUnloadTimeout);
tonUnloadStandstillConfirm(
    IN := (eState = CFF_CONTROLLED_FORCE_UNLOAD)
        AND NOT bStateEntry
        AND bUnloadStandstillQualified,
    PT := stSequenceConfigSnapshot.tUnloadStandstillConfirm);
tonExitRAxisStop(
    IN := (bSafeExitRStopPending OR bUnknownExternalRStopPending
        OR bApproachFaultStopPending)
        AND NOT ((GVL_Status.stFast.udiAcceptedSequenceRCommandId = udiRCommandId)
            AND GVL_Status.stFast.stRAxis.bStandstill),
    PT := stSequenceConfigSnapshot.tRAxisStopTimeout);
tonReturn(
    IN := (eState = CFF_RETURN_LOCAL) OR (eState = CFF_RETURN_REFERENCE),
    PT := stSequenceConfigSnapshot.tReturnTimeout);

IF tonExitRAxisStop.Q THEN
    IF udiFirstFaultId = 0 THEN
        udiFirstFaultId := 16#0000A014;
    END_IF
END_IF

(* One candidate and one complete comparison drive every step R transaction. *)
stCandidateRCommand := stLastPublishedRCommand;
IF ((eState = CFF_STEP1_ENTRY) OR (eState = CFF_STEP2_ENTRY)
    OR (eState = CFF_STEP3_ENTRY)) AND bEntryMotionPermitted THEN
    stCandidateRCommand.bEnable := TRUE;
    stCandidateRCommand.bReset := FALSE;
    stCandidateRCommand.bStop := FALSE;
    stCandidateRCommand.bMoveVelocity := TRUE;
    stCandidateRCommand.rVelocity_rpm :=
        stCycleSnapshot.stProgram.astSteps[nActiveStepProgramIndex].fSetSpeedRpm;
    stCandidateRCommand.rAcceleration_rpm_s := stRAxisProfileSnapshot.fSpeedRampRpmS;
    stCandidateRCommand.rDeceleration_rpm_s := stRAxisProfileSnapshot.fSpeedRampRpmS;
ELSIF eState = CFF_BRAKE_AND_COMPRESSION_RAMP THEN
    stCandidateRCommand.bEnable := TRUE;
    stCandidateRCommand.bReset := FALSE;
    stCandidateRCommand.bStop := TRUE;
    stCandidateRCommand.bMoveVelocity := FALSE;
    stCandidateRCommand.rVelocity_rpm := 0.0;
    stCandidateRCommand.rAcceleration_rpm_s := stRAxisProfileSnapshot.fSpeedRampRpmS;
    stCandidateRCommand.rDeceleration_rpm_s := stRAxisProfileSnapshot.fSpeedRampRpmS;
ELSIF (eState = CFF_CONTROLLED_FORCE_UNLOAD) AND bStateEntry THEN
    stCandidateRCommand.bEnable := TRUE;
    stCandidateRCommand.bReset := FALSE;
    stCandidateRCommand.bStop := TRUE;
    stCandidateRCommand.bMoveVelocity := FALSE;
    stCandidateRCommand.rVelocity_rpm := 0.0;
    stCandidateRCommand.rAcceleration_rpm_s := stRAxisProfileSnapshot.fSpeedRampRpmS;
    stCandidateRCommand.rDeceleration_rpm_s := stRAxisProfileSnapshot.fSpeedRampRpmS;
END_IF
bRCommandPayloadChanged :=
    stCandidateRCommand.bEnable <> stLastPublishedRCommand.bEnable
    OR stCandidateRCommand.bReset <> stLastPublishedRCommand.bReset
    OR stCandidateRCommand.bStop <> stLastPublishedRCommand.bStop
    OR stCandidateRCommand.bMoveVelocity <> stLastPublishedRCommand.bMoveVelocity
    OR stCandidateRCommand.rVelocity_rpm <> stLastPublishedRCommand.rVelocity_rpm
    OR stCandidateRCommand.rAcceleration_rpm_s
        <> stLastPublishedRCommand.rAcceleration_rpm_s
    OR stCandidateRCommand.rDeceleration_rpm_s
        <> stLastPublishedRCommand.rDeceleration_rpm_s;

(* Unique top-level External owner classifier. *)
bExternalProcessState := (eState >= CFF_EXTSETPOINT_PREPARE)
    AND (eState <= CFF_CONTROLLED_FORCE_UNLOAD);
bExternalOwnerHold := ((eState = CFF_EXTSETPOINT_PREPARE)
    OR (eState = CFF_CONTACT_SEARCH)
    OR (eState = CFF_CONTACT_ACCEPT)
    OR (eState = CFF_STEP1_ENTRY)
    OR (eState = CFF_STEP1_RAMP_PROCESS)
    OR (eState = CFF_STEP1_END_CHECK)
    OR (eState = CFF_STEP2_ENTRY)
    OR (eState = CFF_STEP2_RAMP_PROCESS)
    OR (eState = CFF_STEP2_END_CHECK)
    OR (eState = CFF_STEP3_ENTRY)
    OR (eState = CFF_STEP3_RAMP_PROCESS)
    OR (eState = CFF_STEP3_END_CHECK)
    OR (eState = CFF_BRAKE_AND_COMPRESSION_RAMP)
    OR (eState = CFF_STEP4_VALID_FORCE_HOLD)
    OR (eState = CFF_CONTROLLED_FORCE_UNLOAD)
    OR (eState = CFF_EXTSETPOINT_DISABLE))
    AND NOT GVL_Status.stFast.stZExtSetpoint.bReleaseOwner;

(* The complete Force/External and zero-R package is stable for the whole
   External owner lifetime.  State branches repeat the level contract tokens. *)
IF bExternalOwnerHold THEN
    stMotionIntent.stZCommand.bEnable := TRUE;
    stMotionIntent.stZCommand.bReset := FALSE;
    stMotionIntent.stZCommand.bStop := FALSE;
    stMotionIntent.stZCommand.bHome := FALSE;
    stMotionIntent.stZCommand.bMoveAbsolute := FALSE;
    stMotionIntent.stZCommand.bMoveVelocity := FALSE;
    stMotionIntent.stZCommand.bUseExternalSetpoint := TRUE;
    stMotionIntent.stZCommand.rHomePosition_mm := 0.0;
    stMotionIntent.stZCommand.rPosition_mm := 0.0;
    stMotionIntent.stZCommand.rVelocity_mm_s := 0.0;
    stMotionIntent.stZCommand.rAcceleration_mm_s2 := 0.0;
    stMotionIntent.stZCommand.rDeceleration_mm_s2 :=
        stSequenceConfigSnapshot.fStandardMoveDecelerationMmS2;
    stMotionIntent.stZCommand.eOwnerRequest := Z_OWNER_FORCE_PROCESS;
    stMotionIntent.bRAxisProcessRequested := TRUE;
    stMotionIntent.stRCommand.bEnable := TRUE;
    stMotionIntent.stRCommand.bReset := FALSE;
    stMotionIntent.stRCommand.bStop := TRUE;
    stMotionIntent.stRCommand.bMoveVelocity := FALSE;
    stMotionIntent.stRCommand.rVelocity_rpm := 0.0;
    stMotionIntent.stRCommand.rAcceleration_rpm_s := stRAxisProfileSnapshot.fSpeedRampRpmS;
    stMotionIntent.stRCommand.rDeceleration_rpm_s := stRAxisProfileSnapshot.fSpeedRampRpmS;
END_IF

